# B&R Automation Studio project HealthCareDemo
Automation Studio 4.11.1.147; technology packages: mapp6D 1.1.10000, mappFramework 1.0.0, mappMotion 5.18.0, mappView 5.18.0

## Configuration 4PPC70

CPU 4PPC70.0573-20B, AutomationRuntime B4.91, Build 6.3.0, Safety 0.0, Vc V4.72.2

### Task classes (Cpu.sw)
```
Cyclic#1 (cycle 2000 us, tolerance 0 us):
  ConvSyncDe <- (binary)
  WaveDemo <- (binary)
  ConvUnload <- (binary)
  KalmanTes1 <- (binary)
  VariedMovD <- (binary)
  MacroDemo <- (binary)
  KalmanTest <- (binary)
  RoutingDem <- (binary)
  ProcSt2 <- (binary)
  ProcSt1 <- (binary)
  CycChlCfg <- (binary)
  InspectSt <- (binary)
  DofDemo <- (binary)
  ProcessDem <- (binary)
  DanceDemoC <- (binary)
Cyclic#8 (cycle 2000 us):
  RDICore <- Source.Core.RDICore.prg
DataObjects: McAcpSys
NcDataObjects: McDriveLog, AcpParTab
Binaries: udbdef, FWRules, mvLoader, mCoWebSc, TCData, arsvcreg, arflatprv, arcoal, TCLang, iomap, asfw, Role, ashwd, sysconf, arconfig, ashwac, User, TC, AssemConf, LayoutConf, CockpitSet, mcacpdrv, McAcpSim, McProfGen, McMechSys, MotConf, Hierarchy, VaxisConf, GroupConf, MechConf, FeatConf, AxisConf, FileConf, RecConf, Config_1, Config_2, OpcUaSrv, Config, Settings, CfgRecipe, CITT_FileU, CITT_Alarm, CITT_Recip, Config_4, Config_5, Config_3, Config_6, Config_8, Config_9, Config_7, Config_10, TraceConfi
Libraries: operator, runtime, astime, AsIecCon, McAcp6D, McBase, CoTrace, AsZip, FileIO, standard, AsBrStr, MpBase, MpRecipe, sys_lib, MpFile, brsystem, rdiAcp6D, arssl, asusb, dataobj, asmem, asio, asarprof, powerlnk, asepl, asarlog, aruser, McAcpTrak, MpAxis
```

### Hardware
```
4PPC70_0573_20B : 4PPC70.0573-20B v1.5.4.0
  Connector IF2:
    ActivateDevice = 1
    Mode = Manual
    InternetAddress = 192.168.10.10
    SubnetMask = 255.255.255.0
    ActivateSnmp = 2
    DeviceParam = /EDDN=gei
  ConfigurationID = OnsiteDemo_C80
  Simulation = 1
  UserRamSize = 15000
  RemMemSize = 15000
  RemanentGlobalPvSize = 1000
  TimerDeviceType = EPLX2X
  TimerDevice = 1685_CPU.IF1
  TaskClassIdleTime = 2000
  Cyclic1Duration = 2000
  Cyclic1Tolerance = 0
  Cyclic2Duration = 4000
  Cyclic2Tolerance = 4000
  Cyclic3Duration = 8000
  Cyclic3Tolerance = 8000
  Cyclic4Duration = 16000
  Cyclic4Tolerance = 16000
  Cyclic5Duration = 32000
  Cyclic5Tolerance = 32000
  Cyclic6Duration = 64000
  Cyclic6Tolerance = 64000
  Cyclic7Duration = 128000
  Cyclic7Tolerance = 128000
  Cyclic8Duration = 2000
  FileDevice1
  FileDeviceName1 = 6DMacro
  FileDevicePath1 = F:\Macros
  FileDevice2
  FileDeviceName2 = CNC_PrgDir
  FileDevicePath2 = F:/Programs/
  FileDevice3
  FileDeviceName3 = Recipe
  FileDevicePath3 = F:/Recipes/
  FileDevice4
  FileDeviceName4 = TeachFileDev
  FileDevicePath4 = F:/Teach/
  FileDevice5
  FileDeviceName5 = SvMovies
  FileDevicePath5 = F:/SvMovie
  FileDevice6
  FileDeviceName6 = User
  FileDevicePath6 = F:\
  FileDevice7
  FileDeviceName7 = 6DData
  FileDevicePath7 = C:\
  FtpUser1
  FtpUsername1 = bur  // user
  FtpUserPassword1 = kzPdX7T05qFX/2O0oq22KZRISpE2rDw4PeEeBt2Wff8=  // user
  FtpUserSalt1 = NaiTqhR1
  FTPAccessRight1 = 0
  FTPdevice1 = ALL
  ActivateOpcUa = 1
  OpcUaInformationModels_PV_Version = 1
  KeyMappingFile = VC\4PPC70_0573_20B.dis
8YFLM01.0000.00I-1 : 8YFLM01.0000.00I-1 v0.0.0.1
  Supervision = off
```

### IoMap.iom - 4PPC70_0573_20B/IoMap.iom
```iecst
VAR_CONFIG
	Cyclic#1.::gFB.In.Array[0] AT %IW."8YFLM01.0000.00I-1".EPL_FB_IN_0_I2007_S01;
	Cyclic#1.::gFB.In.Array[1] AT %IW."8YFLM01.0000.00I-1".EPL_FB_IN_1_I2007_S02;
	Cyclic#1.::gFB.In.Array[10] AT %IW."8YFLM01.0000.00I-1".EPL_FB_IN_10_I2007_S0B;
	Cyclic#1.::gFB.In.Array[100] AT %IW."8YFLM01.0000.00I-1".EPL_FB_IN_100_I2007_S65;
	Cyclic#1.::gFB.In.Array[101] AT %IW."8YFLM01.0000.00I-1".EPL_FB_IN_101_I2007_S66;
	Cyclic#1.::gFB.In.Array[102] AT %IW."8YFLM01.0000.00I-1".EPL_FB_IN_102_I2007_S67;
	Cyclic#1.::gFB.In.Array[103] AT %IW."8YFLM01.0000.00I-1".EPL_FB_IN_103_I2007_S68;
	Cyclic#1.::gFB.In.Array[104] AT %IW."8YFLM01.0000.00I-1".EPL_FB_IN_104_I2007_S69;
	Cyclic#1.::gFB.In.Array[105] AT %IW."8YFLM01.0000.00I-1".EPL_FB_IN_105_I2007_S6A;
	Cyclic#1.::gFB.In.Array[106] AT %IW."8YFLM01.0000.00I-1".EPL_FB_IN_106_I2007_S6B;
	Cyclic#1.::gFB.In.Array[107] AT %IW."8YFLM01.0000.00I-1".EPL_FB_IN_107_I2007_S6C;
	Cyclic#1.::gFB.In.Array[108] AT %IW."8YFLM01.0000.00I-1".EPL_FB_IN_108_I2007_S6D;
	Cyclic#1.::gFB.In.Array[109] AT %IW."8YFLM01.0000.00I-1".EPL_FB_IN_109_I2007_S6E;
	Cyclic#1.::gFB.In.Array[11] AT %IW."8YFLM01.0000.00I-1".EPL_FB_IN_11_I2007_S0C;
	Cyclic#1.::gFB.In.Array[110] AT %IW."8YFLM01.0000.00I-1".EPL_FB_IN_110_I2007_S6F;
	Cyclic#1.::gFB.In.Array[111] AT %IW."8YFLM01.0000.00I-1".EPL_FB_IN_111_I2007_S70;
	Cyclic#1.::gFB.In.Array[112] AT %IW."8YFLM01.0000.00I-1".EPL_FB_IN_112_I2007_S71;
	Cyclic#1.::gFB.In.Array[113] AT %IW."8YFLM01.0000.00I-1".EPL_FB_IN_113_I2007_S72;
	Cyclic#1.::gFB.In.Array[114] AT %IW."8YFLM01.0000.00I-1".EPL_FB_IN_114_I2007_S73;
	Cyclic#1.::gFB.In.Array[115] AT %IW."8YFLM01.0000.00I-1".EPL_FB_IN_115_I2007_S74;
	Cyclic#1.::gFB.In.Array[116] AT %IW."8YFLM01.0000.00I-1".EPL_FB_IN_116_I2007_S75;
	Cyclic#1.::gFB.In.Array[117] AT %IW."8YFLM01.0000.00I-1".EPL_FB_IN_117_I2007_S76;
	Cyclic#1.::gFB.In.Array[118] AT %IW."8YFLM01.0000.00I-1".EPL_FB_IN_118_I2007_S77;
	Cyclic#1.::gFB.In.Array[119] AT %IW."8YFLM01.0000.00I-1".EPL_FB_IN_119_I2007_S78;
	Cyclic#1.::gFB.In.Array[12] AT %IW."8YFLM01.0000.00I-1".EPL_FB_IN_12_I2007_S0D;
	Cyclic#1.::gFB.In.Array[120] AT %IW."8YFLM01.0000.00I-1".EPL_FB_IN_120_I2007_S79;
	Cyclic#1.::gFB.In.Array[121] AT %IW."8YFLM01.0000.00I-1".EPL_FB_IN_121_I2007_S7A;
	Cyclic#1.::gFB.In.Array[122] AT %IW."8YFLM01.0000.00I-1".EPL_FB_IN_122_I2007_S7B;
	Cyclic#1.::gFB.In.Array[123] AT %IW."8YFLM01.0000.00I-1".EPL_FB_IN_123_I2007_S7C;
	Cyclic#1.::gFB.In.Array[124] AT %IW."8YFLM01.0000.00I-1".EPL_FB_IN_124_I2007_S7D;
	Cyclic#1.::gFB.In.Array[125] AT %IW."8YFLM01.0000.00I-1".EPL_FB_IN_125_I2007_S7E;
	Cyclic#1.::gFB.In.Array[126] AT %IW."8YFLM01.0000.00I-1".EPL_FB_IN_126_I2007_S7F;
	Cyclic#1.::gFB.In.Array[127] AT %IW."8YFLM01.0000.00I-1".EPL_FB_IN_127_I2007_S80;
	Cyclic#1.::gFB.In.Array[128] AT %IW."8YFLM01.0000.00I-1".EPL_FB_IN_128_I2007_S81;
	Cyclic#1.::gFB.In.Array[129] AT %IW."8YFLM01.0000.00I-1".EPL_FB_IN_129_I2007_S82;
	Cyclic#1.::gFB.In.Array[13] AT %IW."8YFLM01.0000.00I-1".EPL_FB_IN_13_I2007_S0E;
	Cyclic#1.::gFB.In.Array[130] AT %IW."8YFLM01.0000.00I-1".EPL_FB_IN_130_I2007_S83;
	Cyclic#1.::gFB.In.Array[131] AT %IW."8YFLM01.0000.00I-1".EPL_FB_IN_131_I2007_S84;
	Cyclic#1.::gFB.In.Array[132] AT %IW."8YFLM01.0000.00I-1".EPL_FB_IN_132_I2007_S85;
	Cyclic#1.::gFB.In.Array[133] AT %IW."8YFLM01.0000.00I-1".EPL_FB_IN_133_I2007_S86;
	Cyclic#1.::gFB.In.Array[134] AT %IW."8YFLM01.0000.00I-1".EPL_FB_IN_134_I2007_S87;
	Cyclic#1.::gFB.In.Array[135] AT %IW."8YFLM01.0000.00I-1".EPL_FB_IN_135_I2007_S88;
	Cyclic#1.::gFB.In.Array[136] AT %IW."8YFLM01.0000.00I-1".EPL_FB_IN_136_I2007_S89;
	Cyclic#1.::gFB.In.Array[137] AT %IW."8YFLM01.0000.00I-1".EPL_FB_IN_137_I2007_S8A;
	Cyclic#1.::gFB.In.Array[138] AT %IW."8YFLM01.0000.00I-1".EPL_FB_IN_138_I2007_S8B;
	Cyclic#1.::gFB.In.Array[139] AT %IW."8YFLM01.0000.00I-1".EPL_FB_IN_139_I2007_S8C;
	Cyclic#1.::gFB.In.Array[14] AT %IW."8YFLM01.0000.00I-1".EPL_FB_IN_14_I2007_S0F;
	Cyclic#1.::gFB.In.Array[140] AT %IW."8YFLM01.0000.00I-1".EPL_FB_IN_140_I2007_S8D;
	Cyclic#1.::gFB.In.Array[141] AT %IW."8YFLM01.0000.00I-1".EPL_FB_IN_141_I2007_S8E;
	Cyclic#1.::gFB.In.Array[142] AT %IW."8YFLM01.0000.00I-1".EPL_FB_IN_142_I2007_S8F;
	Cyclic#1.::gFB.In.Array[143] AT %IW."8YFLM01.0000.00I-1".EPL_FB_IN_143_I2007_S90;
	Cyclic#1.::gFB.In.Array[144] AT %IW."8YFLM01.0000.00I-1".EPL_FB_IN_144_I2007_S91;
	Cyclic#1.::gFB.In.Array[145] AT %IW."8YFLM01.0000.00I-1".EPL_FB_IN_145_I2007_S92;
	Cyclic#1.::gFB.In.Array[146] AT %IW."8YFLM01.0000.00I-1".EPL_FB_IN_146_I2007_S93;
	Cyclic#1.::gFB.In.Array[147] AT %IW."8YFLM01.0000.00I-1".EPL_FB_IN_147_I2007_S94;
	Cyclic#1.::gFB.In.Array[148] AT %IW."8YFLM01.0000.00I-1".EPL_FB_IN_148_I2007_S95;
	Cyclic#1.::gFB.In.Array[149] AT %IW."8YFLM01.0000.00I-1".EPL_FB_IN_149_I2007_S96;
	Cyclic#1.::gFB.In.Array[15] AT %IW."8YFLM01.0000.00I-1".EPL_FB_IN_15_I2007_S10;
	Cyclic#1.::gFB.In.Array[150] AT %IW."8YFLM01.0000.00I-1".EPL_FB_IN_150_I2007_S97;
	Cyclic#1.::gFB.In.Array[151] AT %IW."8YFLM01.0000.00I-1".EPL_FB_IN_151_I2007_S98;
	Cyclic#1.::gFB.In.Array[152] AT %IW."8YFLM01.0000.00I-1".EPL_FB_IN_152_I2007_S99;
	Cyclic#1.::gFB.In.Array[153] AT %IW."8YFLM01.0000.00I-1".EPL_FB_IN_153_I2007_S9A;
	Cyclic#1.::gFB.In.Array[154] AT %IW."8YFLM01.0000.00I-1".EPL_FB_IN_154_I2007_S9B;
	Cyclic#1.::gFB.In.Array[155] AT %IW."8YFLM01.0000.00I-1".EPL_FB_IN_155_I2007_S9C;
	Cyclic#1.::gFB.In.Array[156] AT %IW."8YFLM01.0000.00I-1".EPL_FB_IN_156_I2007_S9D;
	Cyclic#1.::gFB.In.Array[157] AT %IW."8YFLM01.0000.00I-1".EPL_FB_IN_157_I2007_S9E;
	Cyclic#1.::gFB.In.Array[158] AT %IW."8YFLM01.0000.00I-1".EPL_FB_IN_158_I2007_S9F;
	Cyclic#1.::gFB.In.Array[159] AT %IW."8YFLM01.0000.00I-1".EPL_FB_IN_159_I2007_SA0;
	Cyclic#1.::gFB.In.Array[16] AT %IW."8YFLM01.0000.00I-1".EPL_FB_IN_16_I2007_S11;
	Cyclic#1.::gFB.In.Array[160] AT %IW."8YFLM01.0000.00I-1".EPL_FB_IN_160_I2007_SA1;
	Cyclic#1.::gFB.In.Array[161] AT %IW."8YFLM01.0000.00I-1".EPL_FB_IN_161_I2007_SA2;
	Cyclic#1.::gFB.In.Array[162] AT %IW."8YFLM01.0000.00I-1".EPL_FB_IN_162_I2007_SA3;
	Cyclic#1.::gFB.In.Array[163] AT %IW."8YFLM01.0000.00I-1".EPL_FB_IN_163_I2007_SA4;
	Cyclic#1.::gFB.In.Array[164] AT %IW."8YFLM01.0000.00I-1".EPL_FB_IN_164_I2007_SA5;
	Cyclic#1.::gFB.In.Array[165] AT %IW."8YFLM01.0000.00I-1".EPL_FB_IN_165_I2007_SA6;
	Cyclic#1.::gFB.In.Array[166] AT %IW."8YFLM01.0000.00I-1".EPL_FB_IN_166_I2007_SA7;
	Cyclic#1.::gFB.In.Array[167] AT %IW."8YFLM01.0000.00I-1".EPL_FB_IN_167_I2007_SA8;
	Cyclic#1.::gFB.In.Array[168] AT %IW."8YFLM01.0000.00I-1".EPL_FB_IN_168_I2007_SA9;
	Cyclic#1.::gFB.In.Array[169] AT %IW."8YFLM01.0000.00I-1".EPL_FB_IN_169_I2007_SAA;
	Cyclic#1.::gFB.In.Array[17] AT %IW."8YFLM01.0000.00I-1".EPL_FB_IN_17_I2007_S12;
	Cyclic#1.::gFB.In.Array[170] AT %IW."8YFLM01.0000.00I-1".EPL_FB_IN_170_I2007_SAB;
	Cyclic#1.::gFB.In.Array[171] AT %IW."8YFLM01.0000.00I-1".EPL_FB_IN_171_I2007_SAC;
	Cyclic#1.::gFB.In.Array[172] AT %IW."8YFLM01.0000.00I-1".EPL_FB_IN_172_I2007_SAD;
	Cyclic#1.::gFB.In.Array[173] AT %IW."8YFLM01.0000.00I-1".EPL_FB_IN_173_I2007_SAE;
	Cyclic#1.::gFB.In.Array[174] AT %IW."8YFLM01.0000.00I-1".EPL_FB_IN_174_I2007_SAF;
	Cyclic#1.::gFB.In.Array[175] AT %IW."8YFLM01.0000.00I-1".EPL_FB_IN_175_I2007_SB0;
	Cyclic#1.::gFB.In.Array[176] AT %IW."8YFLM01.0000.00I-1".EPL_FB_IN_176_I2007_SB1;
	Cyclic#1.::gFB.In.Array[177] AT %IW."8YFLM01.0000.00I-1".EPL_FB_IN_177_I2007_SB2;
	Cyclic#1.::gFB.In.Array[178] AT %IW."8YFLM01.0000.00I-1".EPL_FB_IN_178_I2007_SB3;
	Cyclic#1.::gFB.In.Array[179] AT %IW."8YFLM01.0000.00I-1".EPL_FB_IN_179_I2007_SB4;
	Cyclic#1.::gFB.In.Array[18] AT %IW."8YFLM01.0000.00I-1".EPL_FB_IN_18_I2007_S13;
	Cyclic#1.::gFB.In.Array[180] AT %IW."8YFLM01.0000.00I-1".EPL_FB_IN_180_I2007_SB5;
	Cyclic#1.::gFB.In.Array[181] AT %IW."8YFLM01.0000.00I-1".EPL_FB_IN_181_I2007_SB6;
	Cyclic#1.::gFB.In.Array[182] AT %IW."8YFLM01.0000.00I-1".EPL_FB_IN_182_I2007_SB7;
	Cyclic#1.::gFB.In.Array[183] AT %IW."8YFLM01.0000.00I-1".EPL_FB_IN_183_I2007_SB8;
	Cyclic#1.::gFB.In.Array[184] AT %IW."8YFLM01.0000.00I-1".EPL_FB_IN_184_I2007_SB9;
	Cyclic#1.::gFB.In.Array[185] AT %IW."8YFLM01.0000.00I-1".EPL_FB_IN_185_I2007_SBA;
	Cyclic#1.::gFB.In.Array[186] AT %IW."8YFLM01.0000.00I-1".EPL_FB_IN_186_I2007_SBB;
	Cyclic#1.::gFB.In.Array[187] AT %IW."8YFLM01.0000.00I-1".EPL_FB_IN_187_I2007_SBC;
	Cyclic#1.::gFB.In.Array[188] AT %IW."8YFLM01.0000.00I-1".EPL_FB_IN_188_I2007_SBD;
	Cyclic#1.::gFB.In.Array[189] AT %IW."8YFLM01.0000.00I-1".EPL_FB_IN_189_I2007_SBE;
	Cyclic#1.::gFB.In.Array[19] AT %IW."8YFLM01.0000.00I-1".EPL_FB_IN_19_I2007_S14;
	Cyclic#1.::gFB.In.Array[190] AT %IW."8YFLM01.0000.00I-1".EPL_FB_IN_190_I2007_SBF;
	Cyclic#1.::gFB.In.Array[191] AT %IW."8YFLM01.0000.00I-1".EPL_FB_IN_191_I2007_SC0;
	Cyclic#1.::gFB.In.Array[192] AT %IW."8YFLM01.0000.00I-1".EPL_FB_IN_192_I2007_SC1;
	Cyclic#1.::gFB.In.Array[193] AT %IW."8YFLM01.0000.00I-1".EPL_FB_IN_193_I2007_SC2;
	Cyclic#1.::gFB.In.Array[194] AT %IW."8YFLM01.0000.00I-1".EPL_FB_IN_194_I2007_SC3;
	Cyclic#1.::gFB.In.Array[195] AT %IW."8YFLM01.0000.00I-1".EPL_FB_IN_195_I2007_SC4;
	Cyclic#1.::gFB.In.Array[196] AT %IW."8YFLM01.0000.00I-1".EPL_FB_IN_196_I2007_SC5;
	Cyclic#1.::gFB.In.Array[197] AT %IW."8YFLM01.0000.00I-1".EPL_FB_IN_197_I2007_SC6;
	Cyclic#1.::gFB.In.Array[198] AT %IW."8YFLM01.0000.00I-1".EPL_FB_IN_198_I2007_SC7;
	Cyclic#1.::gFB.In.Array[199] AT %IW."8YFLM01.0000.00I-1".EPL_FB_IN_199_I2007_SC8;
	Cyclic#1.::gFB.In.Array[2] AT %IW."8YFLM01.0000.00I-1".EPL_FB_IN_2_I2007_S03;
	Cyclic#1.::gFB.In.Array[20] AT %IW."8YFLM01.0000.00I-1".EPL_FB_IN_20_I2007_S15;
	Cyclic#1.::gFB.In.Array[21] AT %IW."8YFLM01.0000.00I-1".EPL_FB_IN_21_I2007_S16;
	Cyclic#1.::gFB.In.Array[22] AT %IW."8YFLM01.0000.00I-1".EPL_FB_IN_22_I2007_S17;
	Cyclic#1.::gFB.In.Array[23] AT %IW."8YFLM01.0000.00I-1".EPL_FB_IN_23_I2007_S18;
	Cyclic#1.::gFB.In.Array[24] AT %IW."8YFLM01.0000.00I-1".EPL_FB_IN_24_I2007_S19;
	Cyclic#1.::gFB.In.Array[25] AT %IW."8YFLM01.0000.00I-1".EPL_FB_IN_25_I2007_S1A;
	Cyclic#1.::gFB.In.Array[26] AT %IW."8YFLM01.0000.00I-1".EPL_FB_IN_26_I2007_S1B;
	Cyclic#1.::gFB.In.Array[27] AT %IW."8YFLM01.0000.00I-1".EPL_FB_IN_27_I2007_S1C;
	Cyclic#1.::gFB.In.Array[28] AT %IW."8YFLM01.0000.00I-1".EPL_FB_IN_28_I2007_S1D;
	Cyclic#1.::gFB.In.Array[29] AT %IW."8YFLM01.0000.00I-1".EPL_FB_IN_29_I2007_S1E;
	Cyclic#1.::gFB.In.Array[3] AT %IW."8YFLM01.0000.00I-1".EPL_FB_IN_3_I2007_S04;
	Cyclic#1.::gFB.In.Array[30] AT %IW."8YFLM01.0000.00I-1".EPL_FB_IN_30_I2007_S1F;
	Cyclic#1.::gFB.In.Array[31] AT %IW."8YFLM01.0000.00I-1".EPL_FB_IN_31_I2007_S20;
	Cyclic#1.::gFB.In.Array[32] AT %IW."8YFLM01.0000.00I-1".EPL_FB_IN_32_I2007_S21;
	Cyclic#1.::gFB.In.Array[33] AT %IW."8YFLM01.0000.00I-1".EPL_FB_IN_33_I2007_S22;
	Cyclic#1.::gFB.In.Array[34] AT %IW."8YFLM01.0000.00I-1".EPL_FB_IN_34_I2007_S23;
	Cyclic#1.::gFB.In.Array[35] AT %IW."8YFLM01.0000.00I-1".EPL_FB_IN_35_I2007_S24;
	Cyclic#1.::gFB.In.Array[36] AT %IW."8YFLM01.0000.00I-1".EPL_FB_IN_36_I2007_S25;
	Cyclic#1.::gFB.In.Array[37] AT %IW."8YFLM01.0000.00I-1".EPL_FB_IN_37_I2007_S26;
	Cyclic#1.::gFB.In.Array[38] AT %IW."8YFLM01.0000.00I-1".EPL_FB_IN_38_I2007_S27;
	Cyclic#1.::gFB.In.Array[39] AT %IW."8YFLM01.0000.00I-1".EPL_FB_IN_39_I2007_S28;
	Cyclic#1.::gFB.In.Array[4] AT %IW."8YFLM01.0000.00I-1".EPL_FB_IN_4_I2007_S05;
	Cyclic#1.::gFB.In.Array[40] AT %IW."8YFLM01.0000.00I-1".EPL_FB_IN_40_I2007_S29;
	Cyclic#1.::gFB.In.Array[41] AT %IW."8YFLM01.0000.00I-1".EPL_FB_IN_41_I2007_S2A;
	Cyclic#1.::gFB.In.Array[42] AT %IW."8YFLM01.0000.00I-1".EPL_FB_IN_42_I2007_S2B;
	Cyclic#1.::gFB.In.Array[43] AT %IW."8YFLM01.0000.00I-1".EPL_FB_IN_43_I2007_S2C;
	Cyclic#1.::gFB.In.Array[44] AT %IW."8YFLM01.0000.00I-1".EPL_FB_IN_44_I2007_S2D;
	Cyclic#1.::gFB.In.Array[45] AT %IW."8YFLM01.0000.00I-1".EPL_FB_IN_45_I2007_S2E;
	Cyclic#1.::gFB.In.Array[46] AT %IW."8YFLM01.0000.00I-1".EPL_FB_IN_46_I2007_S2F;
	Cyclic#1.::gFB.In.Array[47] AT %IW."8YFLM01.0000.00I-1".EPL_FB_IN_47_I2007_S30;
	Cyclic#1.::gFB.In.Array[48] AT %IW."8YFLM01.0000.00I-1".EPL_FB_IN_48_I2007_S31;
	Cyclic#1.::gFB.In.Array[49] AT %IW."8YFLM01.0000.00I-1".EPL_FB_IN_49_I2007_S32;
	Cyclic#1.::gFB.In.Array[5] AT %IW."8YFLM01.0000.00I-1".EPL_FB_IN_5_I2007_S06;
	Cyclic#1.::gFB.In.Array[50] AT %IW."8YFLM01.0000.00I-1".EPL_FB_IN_50_I2007_S33;
	Cyclic#1.::gFB.In.Array[51] AT %IW."8YFLM01.0000.00I-1".EPL_FB_IN_51_I2007_S34;
	Cyclic#1.::gFB.In.Array[52] AT %IW."8YFLM01.0000.00I-1".EPL_FB_IN_52_I2007_S35;
	Cyclic#1.::gFB.In.Array[53] AT %IW."8YFLM01.0000.00I-1".EPL_FB_IN_53_I2007_S36;
	Cyclic#1.::gFB.In.Array[54] AT %IW."8YFLM01.0000.00I-1".EPL_FB_IN_54_I2007_S37;
	Cyclic#1.::gFB.In.Array[55] AT %IW."8YFLM01.0000.00I-1".EPL_FB_IN_55_I2007_S38;
	Cyclic#1.::gFB.In.Array[56] AT %IW."8YFLM01.0000.00I-1".EPL_FB_IN_56_I2007_S39;
	Cyclic#1.::gFB.In.Array[57] AT %IW."8YFLM01.0000.00I-1".EPL_FB_IN_57_I2007_S3A;
	Cyclic#1.::gFB.In.Array[58] AT %IW."8YFLM01.0000.00I-1".EPL_FB_IN_58_I2007_S3B;
	Cyclic#1.::gFB.In.Array[59] AT %IW."8YFLM01.0000.00I-1".EPL_FB_IN_59_I2007_S3C;
	Cyclic#1.::gFB.In.Array[6] AT %IW."8YFLM01.0000.00I-1".EPL_FB_IN_6_I2007_S07;
	Cyclic#1.::gFB.In.Array[60] AT %IW."8YFLM01.0000.00I-1".EPL_FB_IN_60_I2007_S3D;
	Cyclic#1.::gFB.In.Array[61] AT %IW."8YFLM01.0000.00I-1".EPL_FB_IN_61_I2007_S3E;
	Cyclic#1.::gFB.In.Array[62] AT %IW."8YFLM01.0000.00I-1".EPL_FB_IN_62_I2007_S3F;
	Cyclic#1.::gFB.In.Array[63] AT %IW."8YFLM01.0000.00I-1".EPL_FB_IN_63_I2007_S40;
	Cyclic#1.::gFB.In.Array[64] AT %IW."8YFLM01.0000.00I-1".EPL_FB_IN_64_I2007_S41;
	Cyclic#1.::gFB.In.Array[65] AT %IW."8YFLM01.0000.00I-1".EPL_FB_IN_65_I2007_S42;
	Cyclic#1.::gFB.In.Array[66] AT %IW."8YFLM01.0000.00I-1".EPL_FB_IN_66_I2007_S43;
	Cyclic#1.::gFB.In.Array[67] AT %IW."8YFLM01.0000.00I-1".EPL_FB_IN_67_I2007_S44;
	Cyclic#1.::gFB.In.Array[68] AT %IW."8YFLM01.0000.00I-1".EPL_FB_IN_68_I2007_S45;
	Cyclic#1.::gFB.In.Array[69] AT %IW."8YFLM01.0000.00I-1".EPL_FB_IN_69_I2007_S46;
	Cyclic#1.::gFB.In.Array[7] AT %IW."8YFLM01.0000.00I-1".EPL_FB_IN_7_I2007_S08;
	Cyclic#1.::gFB.In.Array[70] AT %IW."8YFLM01.0000.00I-1".EPL_FB_IN_70_I2007_S47;
	Cyclic#1.::gFB.In.Array[71] AT %IW."8YFLM01.0000.00I-1".EPL_FB_IN_71_I2007_S48;
	Cyclic#1.::gFB.In.Array[72] AT %IW."8YFLM01.0000.00I-1".EPL_FB_IN_72_I2007_S49;
	Cyclic#1.::gFB.In.Array[73] AT %IW."8YFLM01.0000.00I-1".EPL_FB_IN_73_I2007_S4A;
	Cyclic#1.::gFB.In.Array[74] AT %IW."8YFLM01.0000.00I-1".EPL_FB_IN_74_I2007_S4B;
	Cyclic#1.::gFB.In.Array[75] AT %IW."8YFLM01.0000.00I-1".EPL_FB_IN_75_I2007_S4C;
	Cyclic#1.::gFB.In.Array[76] AT %IW."8YFLM01.0000.00I-1".EPL_FB_IN_76_I2007_S4D;
	Cyclic#1.::gFB.In.Array[77] AT %IW."8YFLM01.0000.00I-1".EPL_FB_IN_77_I2007_S4E;
	Cyclic#1.::gFB.In.Array[78] AT %IW."8YFLM01.0000.00I-1".EPL_FB_IN_78_I2007_S4F;
	Cyclic#1.::gFB.In.Array[79] AT %IW."8YFLM01.0000.00I-1".EPL_FB_IN_79_I2007_S50;
	Cyclic#1.::gFB.In.Array[8] AT %IW."8YFLM01.0000.00I-1".EPL_FB_IN_8_I2007_S09;
	Cyclic#1.::gFB.In.Array[80] AT %IW."8YFLM01.0000.00I-1".EPL_FB_IN_80_I2007_S51;
	Cyclic#1.::gFB.In.Array[81] AT %IW."8YFLM01.0000.00I-1".EPL_FB_IN_81_I2007_S52;
	Cyclic#1.::gFB.In.Array[82] AT %IW."8YFLM01.0000.00I-1".EPL_FB_IN_82_I2007_S53;
	Cyclic#1.::gFB.In.Array[83] AT %IW."8YFLM01.0000.00I-1".EPL_FB_IN_83_I2007_S54;
	Cyclic#1.::gFB.In.Array[84] AT %IW."8YFLM01.0000.00I-1".EPL_FB_IN_84_I2007_S55;
	Cyclic#1.::gFB.In.Array[85] AT %IW."8YFLM01.0000.00I-1".EPL_FB_IN_85_I2007_S56;
	Cyclic#1.::gFB.In.Array[86] AT %IW."8YFLM01.0000.00I-1".EPL_FB_IN_86_I2007_S57;
	Cyclic#1.::gFB.In.Array[87] AT %IW."8YFLM01.0000.00I-1".EPL_FB_IN_87_I2007_S58;
	Cyclic#1.::gFB.In.Array[88] AT %IW."8YFLM01.0000.00I-1".EPL_FB_IN_88_I2007_S59;
	Cyclic#1.::gFB.In.Array[89] AT %IW."8YFLM01.0000.00I-1".EPL_FB_IN_89_I2007_S5A;
	Cyclic#1.::gFB.In.Array[9] AT %IW."8YFLM01.0000.00I-1".EPL_FB_IN_9_I2007_S0A;
	Cyclic#1.::gFB.In.Array[90] AT %IW."8YFLM01.0000.00I-1".EPL_FB_IN_90_I2007_S5B;
	Cyclic#1.::gFB.In.Array[91] AT %IW."8YFLM01.0000.00I-1".EPL_FB_IN_91_I2007_S5C;
	Cyclic#1.::gFB.In.Array[92] AT %IW."8YFLM01.0000.00I-1".EPL_FB_IN_92_I2007_S5D;
	Cyclic#1.::gFB.In.Array[93] AT %IW."8YFLM01.0000.00I-1".EPL_FB_IN_93_I2007_S5E;
	Cyclic#1.::gFB.In.Array[94] AT %IW."8YFLM01.0000.00I-1".EPL_FB_IN_94_I2007_S5F;
	Cyclic#1.::gFB.In.Array[95] AT %IW."8YFLM01.0000.00I-1".EPL_FB_IN_95_I2007_S60;
	Cyclic#1.::gFB.In.Array[96] AT %IW."8YFLM01.0000.00I-1".EPL_FB_IN_96_I2007_S61;
	Cyclic#1.::gFB.In.Array[97] AT %IW."8YFLM01.0000.00I-1".EPL_FB_IN_97_I2007_S62;
	Cyclic#1.::gFB.In.Array[98] AT %IW."8YFLM01.0000.00I-1".EPL_FB_IN_98_I2007_S63;
	Cyclic#1.::gFB.In.Array[99] AT %IW."8YFLM01.0000.00I-1".EPL_FB_IN_99_I2007_S64;
	Cyclic#1.::gFB.Out.Array[0] AT %QW."8YFLM01.0000.00I-1".EPL_FB_OUT_0_I2008_S01Out;
	Cyclic#1.::gFB.Out.Array[1] AT %QW."8YFLM01.0000.00I-1".EPL_FB_OUT_1_I2008_S02Out;
	Cyclic#1.::gFB.Out.Array[10] AT %QW."8YFLM01.0000.00I-1".EPL_FB_OUT_10_I2008_S0BOut;
	Cyclic#1.::gFB.Out.Array[100] AT %QW."8YFLM01.0000.00I-1".EPL_FB_OUT_100_I2008_S65Out;
	Cyclic#1.::gFB.Out.Array[101] AT %QW."8YFLM01.0000.00I-1".EPL_FB_OUT_101_I2008_S66Out;
	Cyclic#1.::gFB.Out.Array[102] AT %QW."8YFLM01.0000.00I-1".EPL_FB_OUT_102_I2008_S67Out;
	Cyclic#1.::gFB.Out.Array[103] AT %QW."8YFLM01.0000.00I-1".EPL_FB_OUT_103_I2008_S68Out;
	Cyclic#1.::gFB.Out.Array[104] AT %QW."8YFLM01.0000.00I-1".EPL_FB_OUT_104_I2008_S69Out;
	Cyclic#1.::gFB.Out.Array[105] AT %QW."8YFLM01.0000.00I-1".EPL_FB_OUT_105_I2008_S6AOut;
	Cyclic#1.::gFB.Out.Array[106] AT %QW."8YFLM01.0000.00I-1".EPL_FB_OUT_106_I2008_S6BOut;
	Cyclic#1.::gFB.Out.Array[107] AT %QW."8YFLM01.0000.00I-1".EPL_FB_OUT_107_I2008_S6COut;
	Cyclic#1.::gFB.Out.Array[108] AT %QW."8YFLM01.0000.00I-1".EPL_FB_OUT_108_I2008_S6DOut;
	Cyclic#1.::gFB.Out.Array[109] AT %QW."8YFLM01.0000.00I-1".EPL_FB_OUT_109_I2008_S6EOut;
	Cyclic#1.::gFB.Out.Array[11] AT %QW."8YFLM01.0000.00I-1".EPL_FB_OUT_11_I2008_S0COut;
	Cyclic#1.::gFB.Out.Array[110] AT %QW."8YFLM01.0000.00I-1".EPL_FB_OUT_110_I2008_S6FOut;
	Cyclic#1.::gFB.Out.Array[111] AT %QW."8YFLM01.0000.00I-1".EPL_FB_OUT_111_I2008_S70Out;
	Cyclic#1.::gFB.Out.Array[112] AT %QW."8YFLM01.0000.00I-1".EPL_FB_OUT_112_I2008_S71Out;
	Cyclic#1.::gFB.Out.Array[113] AT %QW."8YFLM01.0000.00I-1".EPL_FB_OUT_113_I2008_S72Out;
	Cyclic#1.::gFB.Out.Array[114] AT %QW."8YFLM01.0000.00I-1".EPL_FB_OUT_114_I2008_S73Out;
	Cyclic#1.::gFB.Out.Array[115] AT %QW."8YFLM01.0000.00I-1".EPL_FB_OUT_115_I2008_S74Out;
	Cyclic#1.::gFB.Out.Array[116] AT %QW."8YFLM01.0000.00I-1".EPL_FB_OUT_116_I2008_S75Out;
	Cyclic#1.::gFB.Out.Array[117] AT %QW."8YFLM01.0000.00I-1".EPL_FB_OUT_117_I2008_S76Out;
	Cyclic#1.::gFB.Out.Array[118] AT %QW."8YFLM01.0000.00I-1".EPL_FB_OUT_118_I2008_S77Out;
	Cyclic#1.::gFB.Out.Array[119] AT %QW."8YFLM01.0000.00I-1".EPL_FB_OUT_119_I2008_S78Out;
	Cyclic#1.::gFB.Out.Array[12] AT %QW."8YFLM01.0000.00I-1".EPL_FB_OUT_12_I2008_S0DOut;
	Cyclic#1.::gFB.Out.Array[120] AT %QW."8YFLM01.0000.00I-1".EPL_FB_OUT_120_I2008_S79Out;
	Cyclic#1.::gFB.Out.Array[121] AT %QW."8YFLM01.0000.00I-1".EPL_FB_OUT_121_I2008_S7AOut;
	Cyclic#1.::gFB.Out.Array[122] AT %QW."8YFLM01.0000.00I-1".EPL_FB_OUT_122_I2008_S7BOut;
	Cyclic#1.::gFB.Out.Array[123] AT %QW."8YFLM01.0000.00I-1".EPL_FB_OUT_123_I2008_S7COut;
	Cyclic#1.::gFB.Out.Array[124] AT %QW."8YFLM01.0000.00I-1".EPL_FB_OUT_124_I2008_S7DOut;
	Cyclic#1.::gFB.Out.Array[125] AT %QW."8YFLM01.0000.00I-1".EPL_FB_OUT_125_I2008_S7EOut;
	Cyclic#1.::gFB.Out.Array[126] AT %QW."8YFLM01.0000.00I-1".EPL_FB_OUT_126_I2008_S7FOut;
	Cyclic#1.::gFB.Out.Array[127] AT %QW."8YFLM01.0000.00I-1".EPL_FB_OUT_127_I2008_S80Out;
	Cyclic#1.::gFB.Out.Array[128] AT %QW."8YFLM01.0000.00I-1".EPL_FB_OUT_128_I2008_S81Out;
	Cyclic#1.::gFB.Out.Array[129] AT %QW."8YFLM01.0000.00I-1".EPL_FB_OUT_129_I2008_S82Out;
	Cyclic#1.::gFB.Out.Array[13] AT %QW."8YFLM01.0000.00I-1".EPL_FB_OUT_13_I2008_S0EOut;
	Cyclic#1.::gFB.Out.Array[130] AT %QW."8YFLM01.0000.00I-1".EPL_FB_OUT_130_I2008_S83Out;
	Cyclic#1.::gFB.Out.Array[131] AT %QW."8YFLM01.0000.00I-1".EPL_FB_OUT_131_I2008_S84Out;
	Cyclic#1.::gFB.Out.Array[132] AT %QW."8YFLM01.0000.00I-1".EPL_FB_OUT_132_I2008_S85Out;
	Cyclic#1.::gFB.Out.Array[133] AT %QW."8YFLM01.0000.00I-1".EPL_FB_OUT_133_I2008_S86Out;
	Cyclic#1.::gFB.Out.Array[134] AT %QW."8YFLM01.0000.00I-1".EPL_FB_OUT_134_I2008_S87Out;
	Cyclic#1.::gFB.Out.Array[135] AT %QW."8YFLM01.0000.00I-1".EPL_FB_OUT_135_I2008_S88Out;
	Cyclic#1.::gFB.Out.Array[136] AT %QW."8YFLM01.0000.00I-1".EPL_FB_OUT_136_I2008_S89Out;
	Cyclic#1.::gFB.Out.Array[137] AT %QW."8YFLM01.0000.00I-1".EPL_FB_OUT_137_I2008_S8AOut;
	Cyclic#1.::gFB.Out.Array[138] AT %QW."8YFLM01.0000.00I-1".EPL_FB_OUT_138_I2008_S8BOut;
	Cyclic#1.::gFB.Out.Array[139] AT %QW."8YFLM01.0000.00I-1".EPL_FB_OUT_139_I2008_S8COut;
	Cyclic#1.::gFB.Out.Array[14] AT %QW."8YFLM01.0000.00I-1".EPL_FB_OUT_14_I2008_S0FOut;
	Cyclic#1.::gFB.Out.Array[140] AT %QW."8YFLM01.0000.00I-1".EPL_FB_OUT_140_I2008_S8DOut;
	Cyclic#1.::gFB.Out.Array[141] AT %QW."8YFLM01.0000.00I-1".EPL_FB_OUT_141_I2008_S8EOut;
	Cyclic#1.::gFB.Out.Array[142] AT %QW."8YFLM01.0000.00I-1".EPL_FB_OUT_142_I2008_S8FOut;
	Cyclic#1.::gFB.Out.Array[143] AT %QW."8YFLM01.0000.00I-1".EPL_FB_OUT_143_I2008_S90Out;
	Cyclic#1.::gFB.Out.Array[144] AT %QW."8YFLM01.0000.00I-1".EPL_FB_OUT_144_I2008_S91Out;
	Cyclic#1.::gFB.Out.Array[145] AT %QW."8YFLM01.0000.00I-1".EPL_FB_OUT_145_I2008_S92Out;
	Cyclic#1.::gFB.Out.Array[146] AT %QW."8YFLM01.0000.00I-1".EPL_FB_OUT_146_I2008_S93Out;
	Cyclic#1.::gFB.Out.Array[147] AT %QW."8YFLM01.0000.00I-1".EPL_FB_OUT_147_I2008_S94Out;
	Cyclic#1.::gFB.Out.Array[148] AT %QW."8YFLM01.0000.00I-1".EPL_FB_OUT_148_I2008_S95Out;
	Cyclic#1.::gFB.Out.Array[149] AT %QW."8YFLM01.0000.00I-1".EPL_FB_OUT_149_I2008_S96Out;
	Cyclic#1.::gFB.Out.Array[15] AT %QW."8YFLM01.0000.00I-1".EPL_FB_OUT_15_I2008_S10Out;
	Cyclic#1.::gFB.Out.Array[150] AT %QW."8YFLM01.0000.00I-1".EPL_FB_OUT_150_I2008_S97Out;
	Cyclic#1.::gFB.Out.Array[151] AT %QW."8YFLM01.0000.00I-1".EPL_FB_OUT_151_I2008_S98Out;
	Cyclic#1.::gFB.Out.Array[152] AT %QW."8YFLM01.0000.00I-1".EPL_FB_OUT_152_I2008_S99Out;
	Cyclic#1.::gFB.Out.Array[153] AT %QW."8YFLM01.0000.00I-1".EPL_FB_OUT_153_I2008_S9AOut;
	Cyclic#1.::gFB.Out.Array[154] AT %QW."8YFLM01.0000.00I-1".EPL_FB_OUT_154_I2008_S9BOut;
	Cyclic#1.::gFB.Out.Array[155] AT %QW."8YFLM01.0000.00I-1".EPL_FB_OUT_155_I2008_S9COut;
	Cyclic#1.::gFB.Out.Array[156] AT %QW."8YFLM01.0000.00I-1".EPL_FB_OUT_156_I2008_S9DOut;
	Cyclic#1.::gFB.Out.Array[157] AT %QW."8YFLM01.0000.00I-1".EPL_FB_OUT_157_I2008_S9EOut;
	Cyclic#1.::gFB.Out.Array[158] AT %QW."8YFLM01.0000.00I-1".EPL_FB_OUT_158_I2008_S9FOut;
	Cyclic#1.::gFB.Out.Array[159] AT %QW."8YFLM01.0000.00I-1".EPL_FB_OUT_159_I2008_SA0Out;
	Cyclic#1.::gFB.Out.Array[16] AT %QW."8YFLM01.0000.00I-1".EPL_FB_OUT_16_I2008_S11Out;
	Cyclic#1.::gFB.Out.Array[160] AT %QW."8YFLM01.0000.00I-1".EPL_FB_OUT_160_I2008_SA1Out;
	Cyclic#1.::gFB.Out.Array[161] AT %QW."8YFLM01.0000.00I-1".EPL_FB_OUT_161_I2008_SA2Out;
	Cyclic#1.::gFB.Out.Array[162] AT %QW."8YFLM01.0000.00I-1".EPL_FB_OUT_162_I2008_SA3Out;
	Cyclic#1.::gFB.Out.Array[163] AT %QW."8YFLM01.0000.00I-1".EPL_FB_OUT_163_I2008_SA4Out;
	Cyclic#1.::gFB.Out.Array[164] AT %QW."8YFLM01.0000.00I-1".EPL_FB_OUT_164_I2008_SA5Out;
	Cyclic#1.::gFB.Out.Array[165] AT %QW."8YFLM01.0000.00I-1".EPL_FB_OUT_165_I2008_SA6Out;
	Cyclic#1.::gFB.Out.Array[166] AT %QW."8YFLM01.0000.00I-1".EPL_FB_OUT_166_I2008_SA7Out;
	Cyclic#1.::gFB.Out.Array[167] AT %QW."8YFLM01.0000.00I-1".EPL_FB_OUT_167_I2008_SA8Out;
	Cyclic#1.::gFB.Out.Array[168] AT %QW."8YFLM01.0000.00I-1".EPL_FB_OUT_168_I2008_SA9Out;
	Cyclic#1.::gFB.Out.Array[169] AT %QW."8YFLM01.0000.00I-1".EPL_FB_OUT_169_I2008_SAAOut;
	Cyclic#1.::gFB.Out.Array[17] AT %QW."8YFLM01.0000.00I-1".EPL_FB_OUT_17_I2008_S12Out;
	Cyclic#1.::gFB.Out.Array[170] AT %QW."8YFLM01.0000.00I-1".EPL_FB_OUT_170_I2008_SABOut;
	Cyclic#1.::gFB.Out.Array[171] AT %QW."8YFLM01.0000.00I-1".EPL_FB_OUT_171_I2008_SACOut;
	Cyclic#1.::gFB.Out.Array[172] AT %QW."8YFLM01.0000.00I-1".EPL_FB_OUT_172_I2008_SADOut;
	Cyclic#1.::gFB.Out.Array[173] AT %QW."8YFLM01.0000.00I-1".EPL_FB_OUT_173_I2008_SAEOut;
	Cyclic#1.::gFB.Out.Array[174] AT %QW."8YFLM01.0000.00I-1".EPL_FB_OUT_174_I2008_SAFOut;
	Cyclic#1.::gFB.Out.Array[175] AT %QW."8YFLM01.0000.00I-1".EPL_FB_OUT_175_I2008_SB0Out;
	Cyclic#1.::gFB.Out.Array[176] AT %QW."8YFLM01.0000.00I-1".EPL_FB_OUT_176_I2008_SB1Out;
	Cyclic#1.::gFB.Out.Array[177] AT %QW."8YFLM01.0000.00I-1".EPL_FB_OUT_177_I2008_SB2Out;
	Cyclic#1.::gFB.Out.Array[178] AT %QW."8YFLM01.0000.00I-1".EPL_FB_OUT_178_I2008_SB3Out;
	Cyclic#1.::gFB.Out.Array[179] AT %QW."8YFLM01.0000.00I-1".EPL_FB_OUT_179_I2008_SB4Out;
	Cyclic#1.::gFB.Out.Array[18] AT %QW."8YFLM01.0000.00I-1".EPL_FB_OUT_18_I2008_S13Out;
	Cyclic#1.::gFB.Out.Array[180] AT %QW."8YFLM01.0000.00I-1".EPL_FB_OUT_180_I2008_SB5Out;
	Cyclic#1.::gFB.Out.Array[181] AT %QW."8YFLM01.0000.00I-1".EPL_FB_OUT_181_I2008_SB6Out;
	Cyclic#1.::gFB.Out.Array[182] AT %QW."8YFLM01.0000.00I-1".EPL_FB_OUT_182_I2008_SB7Out;
	Cyclic#1.::gFB.Out.Array[183] AT %QW."8YFLM01.0000.00I-1".EPL_FB_OUT_183_I2008_SB8Out;
	Cyclic#1.::gFB.Out.Array[184] AT %QW."8YFLM01.0000.00I-1".EPL_FB_OUT_184_I2008_SB9Out;
	Cyclic#1.::gFB.Out.Array[185] AT %QW."8YFLM01.0000.00I-1".EPL_FB_OUT_185_I2008_SBAOut;
	Cyclic#1.::gFB.Out.Array[186] AT %QW."8YFLM01.0000.00I-1".EPL_FB_OUT_186_I2008_SBBOut;
	Cyclic#1.::gFB.Out.Array[187] AT %QW."8YFLM01.0000.00I-1".EPL_FB_OUT_187_I2008_SBCOut;
	Cyclic#1.::gFB.Out.Array[188] AT %QW."8YFLM01.0000.00I-1".EPL_FB_OUT_188_I2008_SBDOut;
	Cyclic#1.::gFB.Out.Array[189] AT %QW."8YFLM01.0000.00I-1".EPL_FB_OUT_189_I2008_SBEOut;
	Cyclic#1.::gFB.Out.Array[19] AT %QW."8YFLM01.0000.00I-1".EPL_FB_OUT_19_I2008_S14Out;
	Cyclic#1.::gFB.Out.Array[190] AT %QW."8YFLM01.0000.00I-1".EPL_FB_OUT_190_I2008_SBFOut;
	Cyclic#1.::gFB.Out.Array[191] AT %QW."8YFLM01.0000.00I-1".EPL_FB_OUT_191_I2008_SC0Out;
	Cyclic#1.::gFB.Out.Array[192] AT %QW."8YFLM01.0000.00I-1".EPL_FB_OUT_192_I2008_SC1Out;
	Cyclic#1.::gFB.Out.Array[193] AT %QW."8YFLM01.0000.00I-1".EPL_FB_OUT_193_I2008_SC2Out;
	Cyclic#1.::gFB.Out.Array[194] AT %QW."8YFLM01.0000.00I-1".EPL_FB_OUT_194_I2008_SC3Out;
	Cyclic#1.::gFB.Out.Array[195] AT %QW."8YFLM01.0000.00I-1".EPL_FB_OUT_195_I2008_SC4Out;
	Cyclic#1.::gFB.Out.Array[196] AT %QW."8YFLM01.0000.00I-1".EPL_FB_OUT_196_I2008_SC5Out;
	Cyclic#1.::gFB.Out.Array[197] AT %QW."8YFLM01.0000.00I-1".EPL_FB_OUT_197_I2008_SC6Out;
	Cyclic#1.::gFB.Out.Array[198] AT %QW."8YFLM01.0000.00I-1".EPL_FB_OUT_198_I2008_SC7Out;
	Cyclic#1.::gFB.Out.Array[199] AT %QW."8YFLM01.0000.00I-1".EPL_FB_OUT_199_I2008_SC8Out;
	Cyclic#1.::gFB.Out.Array[2] AT %QW."8YFLM01.0000.00I-1".EPL_FB_OUT_2_I2008_S03Out;
	Cyclic#1.::gFB.Out.Array[20] AT %QW."8YFLM01.0000.00I-1".EPL_FB_OUT_20_I2008_S15Out;
	Cyclic#1.::gFB.Out.Array[21] AT %QW."8YFLM01.0000.00I-1".EPL_FB_OUT_21_I2008_S16Out;
	Cyclic#1.::gFB.Out.Array[22] AT %QW."8YFLM01.0000.00I-1".EPL_FB_OUT_22_I2008_S17Out;
	Cyclic#1.::gFB.Out.Array[23] AT %QW."8YFLM01.0000.00I-1".EPL_FB_OUT_23_I2008_S18Out;
	Cyclic#1.::gFB.Out.Array[24] AT %QW."8YFLM01.0000.00I-1".EPL_FB_OUT_24_I2008_S19Out;
	Cyclic#1.::gFB.Out.Array[25] AT %QW."8YFLM01.0000.00I-1".EPL_FB_OUT_25_I2008_S1AOut;
	Cyclic#1.::gFB.Out.Array[26] AT %QW."8YFLM01.0000.00I-1".EPL_FB_OUT_26_I2008_S1BOut;
	Cyclic#1.::gFB.Out.Array[27] AT %QW."8YFLM01.0000.00I-1".EPL_FB_OUT_27_I2008_S1COut;
	Cyclic#1.::gFB.Out.Array[28] AT %QW."8YFLM01.0000.00I-1".EPL_FB_OUT_28_I2008_S1DOut;
	Cyclic#1.::gFB.Out.Array[29] AT %QW."8YFLM01.0000.00I-1".EPL_FB_OUT_29_I2008_S1EOut;
	Cyclic#1.::gFB.Out.Array[3] AT %QW."8YFLM01.0000.00I-1".EPL_FB_OUT_3_I2008_S04Out;
	Cyclic#1.::gFB.Out.Array[30] AT %QW."8YFLM01.0000.00I-1".EPL_FB_OUT_30_I2008_S1FOut;
	Cyclic#1.::gFB.Out.Array[31] AT %QW."8YFLM01.0000.00I-1".EPL_FB_OUT_31_I2008_S20Out;
	Cyclic#1.::gFB.Out.Array[32] AT %QW."8YFLM01.0000.00I-1".EPL_FB_OUT_32_I2008_S21Out;
	Cyclic#1.::gFB.Out.Array[33] AT %QW."8YFLM01.0000.00I-1".EPL_FB_OUT_33_I2008_S22Out;
	Cyclic#1.::gFB.Out.Array[34] AT %QW."8YFLM01.0000.00I-1".EPL_FB_OUT_34_I2008_S23Out;
	Cyclic#1.::gFB.Out.Array[35] AT %QW."8YFLM01.0000.00I-1".EPL_FB_OUT_35_I2008_S24Out;
	Cyclic#1.::gFB.Out.Array[36] AT %QW."8YFLM01.0000.00I-1".EPL_FB_OUT_36_I2008_S25Out;
	Cyclic#1.::gFB.Out.Array[37] AT %QW."8YFLM01.0000.00I-1".EPL_FB_OUT_37_I2008_S26Out;
	Cyclic#1.::gFB.Out.Array[38] AT %QW."8YFLM01.0000.00I-1".EPL_FB_OUT_38_I2008_S27Out;
	Cyclic#1.::gFB.Out.Array[39] AT %QW."8YFLM01.0000.00I-1".EPL_FB_OUT_39_I2008_S28Out;
	Cyclic#1.::gFB.Out.Array[4] AT %QW."8YFLM01.0000.00I-1".EPL_FB_OUT_4_I2008_S05Out;
	Cyclic#1.::gFB.Out.Array[40] AT %QW."8YFLM01.0000.00I-1".EPL_FB_OUT_40_I2008_S29Out;
	Cyclic#1.::gFB.Out.Array[41] AT %QW."8YFLM01.0000.00I-1".EPL_FB_OUT_41_I2008_S2AOut;
	Cyclic#1.::gFB.Out.Array[42] AT %QW."8YFLM01.0000.00I-1".EPL_FB_OUT_42_I2008_S2BOut;
	Cyclic#1.::gFB.Out.Array[43] AT %QW."8YFLM01.0000.00I-1".EPL_FB_OUT_43_I2008_S2COut;
	Cyclic#1.::gFB.Out.Array[44] AT %QW."8YFLM01.0000.00I-1".EPL_FB_OUT_44_I2008_S2DOut;
	Cyclic#1.::gFB.Out.Array[45] AT %QW."8YFLM01.0000.00I-1".EPL_FB_OUT_45_I2008_S2EOut;
	Cyclic#1.::gFB.Out.Array[46] AT %QW."8YFLM01.0000.00I-1".EPL_FB_OUT_46_I2008_S2FOut;
	Cyclic#1.::gFB.Out.Array[47] AT %QW."8YFLM01.0000.00I-1".EPL_FB_OUT_47_I2008_S30Out;
	Cyclic#1.::gFB.Out.Array[48] AT %QW."8YFLM01.0000.00I-1".EPL_FB_OUT_48_I2008_S31Out;
	Cyclic#1.::gFB.Out.Array[49] AT %QW."8YFLM01.0000.00I-1".EPL_FB_OUT_49_I2008_S32Out;
	Cyclic#1.::gFB.Out.Array[5] AT %QW."8YFLM01.0000.00I-1".EPL_FB_OUT_5_I2008_S06Out;
	Cyclic#1.::gFB.Out.Array[50] AT %QW."8YFLM01.0000.00I-1".EPL_FB_OUT_50_I2008_S33Out;
	Cyclic#1.::gFB.Out.Array[51] AT %QW."8YFLM01.0000.00I-1".EPL_FB_OUT_51_I2008_S34Out;
	Cyclic#1.::gFB.Out.Array[52] AT %QW."8YFLM01.0000.00I-1".EPL_FB_OUT_52_I2008_S35Out;
	Cyclic#1.::gFB.Out.Array[53] AT %QW."8YFLM01.0000.00I-1".EPL_FB_OUT_53_I2008_S36Out;
	Cyclic#1.::gFB.Out.Array[54] AT %QW."8YFLM01.0000.00I-1".EPL_FB_OUT_54_I2008_S37Out;
	Cyclic#1.::gFB.Out.Array[55] AT %QW."8YFLM01.0000.00I-1".EPL_FB_OUT_55_I2008_S38Out;
	Cyclic#1.::gFB.Out.Array[56] AT %QW."8YFLM01.0000.00I-1".EPL_FB_OUT_56_I2008_S39Out;
	Cyclic#1.::gFB.Out.Array[57] AT %QW."8YFLM01.0000.00I-1".EPL_FB_OUT_57_I2008_S3AOut;
	Cyclic#1.::gFB.Out.Array[58] AT %QW."8YFLM01.0000.00I-1".EPL_FB_OUT_58_I2008_S3BOut;
	Cyclic#1.::gFB.Out.Array[59] AT %QW."8YFLM01.0000.00I-1".EPL_FB_OUT_59_I2008_S3COut;
	Cyclic#1.::gFB.Out.Array[6] AT %QW."8YFLM01.0000.00I-1".EPL_FB_OUT_6_I2008_S07Out;
	Cyclic#1.::gFB.Out.Array[60] AT %QW."8YFLM01.0000.00I-1".EPL_FB_OUT_60_I2008_S3DOut;
	Cyclic#1.::gFB.Out.Array[61] AT %QW."8YFLM01.0000.00I-1".EPL_FB_OUT_61_I2008_S3EOut;
	Cyclic#1.::gFB.Out.Array[62] AT %QW."8YFLM01.0000.00I-1".EPL_FB_OUT_62_I2008_S3FOut;
	Cyclic#1.::gFB.Out.Array[63] AT %QW."8YFLM01.0000.00I-1".EPL_FB_OUT_63_I2008_S40Out;
	Cyclic#1.::gFB.Out.Array[64] AT %QW."8YFLM01.0000.00I-1".EPL_FB_OUT_64_I2008_S41Out;
	Cyclic#1.::gFB.Out.Array[65] AT %QW."8YFLM01.0000.00I-1".EPL_FB_OUT_65_I2008_S42Out;
	Cyclic#1.::gFB.Out.Array[66] AT %QW."8YFLM01.0000.00I-1".EPL_FB_OUT_66_I2008_S43Out;
	Cyclic#1.::gFB.Out.Array[67] AT %QW."8YFLM01.0000.00I-1".EPL_FB_OUT_67_I2008_S44Out;
	Cyclic#1.::gFB.Out.Array[68] AT %QW."8YFLM01.0000.00I-1".EPL_FB_OUT_68_I2008_S45Out;
	Cyclic#1.::gFB.Out.Array[69] AT %QW."8YFLM01.0000.00I-1".EPL_FB_OUT_69_I2008_S46Out;
	Cyclic#1.::gFB.Out.Array[7] AT %QW."8YFLM01.0000.00I-1".EPL_FB_OUT_7_I2008_S08Out;
	Cyclic#1.::gFB.Out.Array[70] AT %QW."8YFLM01.0000.00I-1".EPL_FB_OUT_70_I2008_S47Out;
	Cyclic#1.::gFB.Out.Array[71] AT %QW."8YFLM01.0000.00I-1".EPL_FB_OUT_71_I2008_S48Out;
	Cyclic#1.::gFB.Out.Array[72] AT %QW."8YFLM01.0000.00I-1".EPL_FB_OUT_72_I2008_S49Out;
	Cyclic#1.::gFB.Out.Array[73] AT %QW."8YFLM01.0000.00I-1".EPL_FB_OUT_73_I2008_S4AOut;
	Cyclic#1.::gFB.Out.Array[74] AT %QW."8YFLM01.0000.00I-1".EPL_FB_OUT_74_I2008_S4BOut;
	Cyclic#1.::gFB.Out.Array[75] AT %QW."8YFLM01.0000.00I-1".EPL_FB_OUT_75_I2008_S4COut;
	Cyclic#1.::gFB.Out.Array[76] AT %QW."8YFLM01.0000.00I-1".EPL_FB_OUT_76_I2008_S4DOut;
	Cyclic#1.::gFB.Out.Array[77] AT %QW."8YFLM01.0000.00I-1".EPL_FB_OUT_77_I2008_S4EOut;
	Cyclic#1.::gFB.Out.Array[78] AT %QW."8YFLM01.0000.00I-1".EPL_FB_OUT_78_I2008_S4FOut;
	Cyclic#1.::gFB.Out.Array[79] AT %QW."8YFLM01.0000.00I-1".EPL_FB_OUT_79_I2008_S50Out;
	Cyclic#1.::gFB.Out.Array[8] AT %QW."8YFLM01.0000.00I-1".EPL_FB_OUT_8_I2008_S09Out;
	Cyclic#1.::gFB.Out.Array[80] AT %QW."8YFLM01.0000.00I-1".EPL_FB_OUT_80_I2008_S51Out;
	Cyclic#1.::gFB.Out.Array[81] AT %QW."8YFLM01.0000.00I-1".EPL_FB_OUT_81_I2008_S52Out;
	Cyclic#1.::gFB.Out.Array[82] AT %QW."8YFLM01.0000.00I-1".EPL_FB_OUT_82_I2008_S53Out;
	Cyclic#1.::gFB.Out.Array[83] AT %QW."8YFLM01.0000.00I-1".EPL_FB_OUT_83_I2008_S54Out;
	Cyclic#1.::gFB.Out.Array[84] AT %QW."8YFLM01.0000.00I-1".EPL_FB_OUT_84_I2008_S55Out;
	Cyclic#1.::gFB.Out.Array[85] AT %QW."8YFLM01.0000.00I-1".EPL_FB_OUT_85_I2008_S56Out;
	Cyclic#1.::gFB.Out.Array[86] AT %QW."8YFLM01.0000.00I-1".EPL_FB_OUT_86_I2008_S57Out;
	Cyclic#1.::gFB.Out.Array[87] AT %QW."8YFLM01.0000.00I-1".EPL_FB_OUT_87_I2008_S58Out;
	Cyclic#1.::gFB.Out.Array[88] AT %QW."8YFLM01.0000.00I-1".EPL_FB_OUT_88_I2008_S59Out;
	Cyclic#1.::gFB.Out.Array[89] AT %QW."8YFLM01.0000.00I-1".EPL_FB_OUT_89_I2008_S5AOut;
	Cyclic#1.::gFB.Out.Array[9] AT %QW."8YFLM01.0000.00I-1".EPL_FB_OUT_9_I2008_S0AOut;
	Cyclic#1.::gFB.Out.Array[90] AT %QW."8YFLM01.0000.00I-1".EPL_FB_OUT_90_I2008_S5BOut;
	Cyclic#1.::gFB.Out.Array[91] AT %QW."8YFLM01.0000.00I-1".EPL_FB_OUT_91_I2008_S5COut;
	Cyclic#1.::gFB.Out.Array[92] AT %QW."8YFLM01.0000.00I-1".EPL_FB_OUT_92_I2008_S5DOut;
	Cyclic#1.::gFB.Out.Array[93] AT %QW."8YFLM01.0000.00I-1".EPL_FB_OUT_93_I2008_S5EOut;
	Cyclic#1.::gFB.Out.Array[94] AT %QW."8YFLM01.0000.00I-1".EPL_FB_OUT_94_I2008_S5FOut;
	Cyclic#1.::gFB.Out.Array[95] AT %QW."8YFLM01.0000.00I-1".EPL_FB_OUT_95_I2008_S60Out;
	Cyclic#1.::gFB.Out.Array[96] AT %QW."8YFLM01.0000.00I-1".EPL_FB_OUT_96_I2008_S61Out;
	Cyclic#1.::gFB.Out.Array[97] AT %QW."8YFLM01.0000.00I-1".EPL_FB_OUT_97_I2008_S62Out;
	Cyclic#1.::gFB.Out.Array[98] AT %QW."8YFLM01.0000.00I-1".EPL_FB_OUT_98_I2008_S63Out;
	Cyclic#1.::gFB.Out.Array[99] AT %QW."8YFLM01.0000.00I-1".EPL_FB_OUT_99_I2008_S64Out;
END_VAR
```

### AssemConf.assembly6d - 4PPC70_0573_20B/mapp6D/AssemConf.assembly6d
```
Element g6dAssembly (Type=assembly6d)
  Simulation6D = SimOn
  Shuttles:
    MaxShuttleCount = 2
    ShuttleIDMode = RealTimeID
    DefaultPosition:
      DefZ = 1.0
      DefRx = 0
      DefRy = 0
      DefRz = 0
    Limits:
      InPlaneLimits:
        InPlaneVelLim = 1.0
        InPlaneAccLim = 10.0
        InPlaneEmergDec = 10.0
      ShortAxLim:
        ShortAxAccLim:
          AccZLim = 10.0
          AccRxLim = 10.0
          AccRyLim = 10.0
          AccRzLim = 10.0
        ShortAxVelLim:
          VelZLim = 0.15
          VelRxLim = 0.1
          VelRyLim = 0.1
          VelRzLim = 0.3
  CyclicChannel6D:
    ReadChannel:
      Xaxis = TRUE
      Yaxis = TRUE
      Zaxis = TRUE
      Rxaxis = TRUE
      Ryaxis = TRUE
      Rzaxis = TRUE
  Fieldbus6D:
    SyncMode6D = ExternalPlkSync
    NodeNumber = 101
  IOMapp:
    Input = ::gFB.In
    Output = ::gFB.Out
  Layout:
    Layout6D[1] = Layout6D_1
  Visualization:
    MonitoringPv = ::gAssemblyMon
    VisPv
    ProcessingTaskClass = 2
```

### LayoutConf.layout6d - 4PPC70_0573_20B/mapp6D/LayoutConf.layout6d
```
Element Layout6D_1 (Type=layout6d)
  Segments:
    SegRow = 1
    SegCol = 2
    Segment[1]:
      X = 0
      Y = 0
      Name
      IsMaster = True
    Segment[2]:
      X = 1
      Y = 0
      Name
      IsMaster = False
```

## Configuration X20CP1685

CPU X20CP1685, AutomationRuntime B4.91, Build 6.3.0, Safety 0.0, Vc V4.72.2

### Task classes (Cpu.sw)
```
Cyclic#1 (cycle 2000 us, tolerance 0 us):
  Acp6DCtrl <- Source.Core.Acp6DCtrl.prg
  ConvSyncDe <- (binary)
  WaveDemo <- (binary)
  ConvUnload <- (binary)
  KalmanTes1 <- (binary)
  VariedMovD <- (binary)
  MacroDemo <- (binary)
  KalmanTest <- (binary)
  RoutingDem <- (binary)
  ProcSt2 <- (binary)
  ProcSt1 <- (binary)
  CycChlCfg <- (binary)
  InspectSt <- (binary)
  DofDemo <- (binary)
  ProcessDem <- (binary)
  DanceDemoC <- (binary)
Cyclic#2 (cycle 4000 us, tolerance 4000 us):
  Program <- Source.Core.Program.prg
  RoutingDef <- Source.Core.RoutingDefinitions.prg
  PipetteSta <- Source.Core.PipetteStations.prg
  Stations <- Source.Core.Stations.prg
  DyeTipStat <- Source.Core.DyeTipStations.prg
Cyclic#4 (cycle 16000 us, tolerance 16000 us):
  Main <- Source.Core.Main.prg
Cyclic#8 (cycle 2000 us):
  RDICore <- Source.Core.RDICore.prg [disabled]
  BuildVer <- Source.BuildVersion.BuildVer.prg
  Vis <- Source.ScnViewer.Vis.prg
DataObjects: McAcpSys
NcDataObjects: mcdrivelog, AcpParTab
Binaries: FWRules, mvLoader, udbdef, TCLang, TCData, arcoal, arsvcreg, arflatprv, iomap, asfw, Role, ashwd, sysconf, arconfig, ashwac, User, TC, AssemConf, LayoutConf, mCoWebSc, CockpitSet, mcacpdrv, McAcpSim, McProfGen, McMechSys, MotConf, Hierarchy, VaxisConf, GroupConf, MechConf, FeatConf, AxisConf, FileConf, RecConf, Config_1, Config_2, OpcUaSrv, Config, Settings, CfgRecipe, CITT_FileU, CITT_Alarm, CITT_Recip, Config_4, Config_5, Config_3, Config_6, Config_8, Config_9, Config_7, Config_10, TraceConfi
Libraries: Acp6dHlpr, McBase, McAcp6D, AsSem, ArEventLog, runtime, Router6D, StnLogic, arssl, fileio, standard, astime, asieccon, asbrstr, mpbase, sys_lib, dataobj, asmem, asio, asarprof, powerlnk, asepl, asarlog, aruser, McAcpTrak, MpAxis
```

### Hardware
```
8YFLM01.0000.00I-1 : 8YFLM01.0000.00I-1 v0.0.0.1  [PLK1 -> X20CP1685.IF3 (NodeNumber=101) [Cable Type=PowerlinkCable, Length=10, Version=1.0.0.3]]
  Supervision = off
X20CP1685 : X20CP1685 v1.4.0.0
  Connector IF2:
    ActivateDevice = 1
    Mode = Manual
    InternetAddress = 192.168.10.81
    SubnetMask = 255.255.255.0
    ActivateSnmp = 2
  Connector IF3:
    CycleTime = 1000
  ConfigurationID = OnsiteDemo_C80
  TimerDeviceType = EPLX2X
  TimerDevice = X20CP1685.IF3
  TaskClassIdleTime = 2000
  Cyclic1Duration = 2000
  Cyclic1Tolerance = 0
  Cyclic2Duration = 4000
  Cyclic2Tolerance = 4000
  Cyclic3Duration = 8000
  Cyclic3Tolerance = 8000
  Cyclic4Duration = 16000
  Cyclic4Tolerance = 16000
  Cyclic5Duration = 32000
  Cyclic5Tolerance = 32000
  Cyclic6Duration = 64000
  Cyclic6Tolerance = 64000
  Cyclic7Duration = 128000
  Cyclic7Tolerance = 128000
  Cyclic8Duration = 2000
  FileDevice1
  FileDeviceName1 = 6DMacro
  FileDevicePath1 = F:\Macros
  FileDevice2
  FileDeviceName2 = CNC_PrgDir
  FileDevicePath2 = F:/Programs/
  FileDevice3
  FileDeviceName3 = Recipe
  FileDevicePath3 = F:/Recipes/
  FileDevice4
  FileDeviceName4 = TeachFileDev
  FileDevicePath4 = F:/Teach/
  FileDevice5
  FileDeviceName5 = SvMovies
  FileDevicePath5 = F:/SvMovie
  FileDevice6
  FileDeviceName6 = User
  FileDevicePath6 = F:\
  FileDevice7
  FileDeviceName7 = 6DData
  FileDevicePath7 = C:\
  FtpUser1
  FtpUsername1 = bur  // user
  FtpUserPassword1 = kzPdX7T05qFX/2O0oq22KZRISpE2rDw4PeEeBt2Wff8=  // user
  FtpUserSalt1 = NaiTqhR1
  FTPAccessRight1 = 0
  FTPdevice1 = ALL
  ActivateOpcUa = 1
  OpcUaInformationModels_PV_Version = 1
```

### AssemConf.assembly6d - X20CP1685/mapp6D/AssemConf.assembly6d
```
Element g6dAssembly (Type=assembly6d)
  Simulation6D = SimOn
  Shuttles:
    MaxShuttleCount = 5
    ShuttleIDMode = RealTimeID
    DefaultPosition:
      DefZ = 1.0
      DefRx = 0
      DefRy = 0
      DefRz = 0
    Limits:
      InPlaneLimits:
        InPlaneVelLim = 1.0
        InPlaneAccLim = 10.0
        InPlaneEmergDec = 10.0
      ShortAxLim:
        ShortAxAccLim:
          AccZLim = 10.0
          AccRxLim = 10.0
          AccRyLim = 10.0
          AccRzLim = 10.0
        ShortAxVelLim:
          VelZLim = 0.15
          VelRxLim = 0.1
          VelRyLim = 0.1
          VelRzLim = 0.3
  CyclicChannel6D:
    ReadChannel:
      Xaxis = TRUE
      Yaxis = TRUE
      Zaxis = TRUE
      Rxaxis = TRUE
      Ryaxis = TRUE
      Rzaxis = TRUE
  Fieldbus6D:
    SyncMode6D = ExternalPlkSync
    NodeNumber = 101
  IOMapp:
    Input = ::gFB.In
    Output = ::gFB.Out
  Layout:
    Layout6D[1] = Layout6D_1
  Visualization:
    MonitoringPv
    VisPv
    ProcessingTaskClass = 4
```

### LayoutConf.layout6d - X20CP1685/mapp6D/LayoutConf.layout6d
```
Element Layout6D_1 (Type=layout6d)
  Segments:
    SegRow = 3
    SegCol = 3
    Segment[1]:
      X = 0
      Y = 0
      Name
      IsMaster = True
    Segment[2]:
      X = 0
      Y = 1
      Name
      IsMaster = False
    Segment[3]:
      X = 0
      Y = 2
      Name
      IsMaster = False
    Segment[4]:
      X = 1
      Y = 0
      Name
      IsMaster = False
    Segment[5]:
      X = 1
      Y = 1
      Name
      IsMaster = False
    Segment[6]:
      X = 1
      Y = 2
      Name
      IsMaster = False
    Segment[7]:
      X = 2
      Y = 1
      Name
      IsMaster = False
```

## Logical view

Binary libraries used (declarations not repeated): operator, runtime, astime, AsIecCon, AsZip, FileIO, standard, AsBrStr, sys_lib, brsystem, MpFile, MpBase, CoTrace, MpRecipe, AsSem, ArEventLog, McBase 5.17.9, McAcp6D 1.01.9

### Global.typ - Global data types
```iecst
TYPE
	gFBType : 	STRUCT  (*6D Interfaces*)
		In : Mc6DControllerFBIOType; (*Inputs*)
		Out : Mc6DControllerFBIOType; (*Outputs*)
	END_STRUCT;
END_TYPE

(************************* Main If Typ*)

TYPE
	MainIfTyp : 	STRUCT
		Cmd : MainIfCmdTyp;
		Par : USINT;
		Sts : USINT;
	END_STRUCT;
	MainIfCmdTyp : 	STRUCT
		Power : BOOL;
		Run : BOOL;
		ErrorReset : BOOL;
	END_STRUCT;
	SystemRecipeIfTyp : 	STRUCT
		DefaultVel : REAL;
		DefaultAccel : REAL;
		DefaultWaitTime : UDINT;
		StartupPars : StartupPars;
		WellRecipe : ARRAY[0..1]OF FillRecipeTyp;
		PipettePars : PipettePars;
	END_STRUCT;
	StartupPars : 	STRUCT
		MoveAsyncPars : McAcp6DMoveInPlaneAsyncParType;
	END_STRUCT;
	PipettePars : 	STRUCT
		HomePosition : REAL;
		Vel : REAL;
		SampleDistance : REAL;
		WellDistance : REAL;
	END_STRUCT;
END_TYPE

(************************* Acp6D Types*)

TYPE
	Acp6DIfTyp : 	STRUCT
		Cmd : Acp6DCmdsTyp;
		Par : Acp6DParTyp;
		Sts : Acp6DStsTyp;
	END_STRUCT;
	Acp6DCmdsTyp : 	STRUCT
		Power : BOOL;
		Reset : BOOL;
		ResetInfo : BOOL;
	END_STRUCT;
	Acp6DParTyp : 	STRUCT
		ShuttleCount : USINT;
		Asm : Mc6DAssemblyType;
	END_STRUCT;
	Acp6DStsTyp : 	STRUCT
		Error : BOOL;
		AssemblyInfo : McAcp6DAsmGetInfoType;
		AssemblyDisabled : BOOL;
		AssemblyReady : BOOL;
		AssemblyHoming : BOOL;
		AssemblyStopping : BOOL;
		AssemblyStartup : BOOL;
		AssemblyErrorStop : BOOL;
	END_STRUCT;
END_TYPE

(************************** Shuttle If Types*)

TYPE
	ShuttleIfTyp : 	STRUCT
		Cmd : ShuttleIfCmdTyp;
		Par : ShuttleIfParTyp;
		Cfg : ShuttleIfCfgTyp;
		Sts : ShuttleIfStsTyp;
	END_STRUCT;
	ShuttleIfCmdTyp : 	STRUCT
		Reset : BOOL;
	END_STRUCT;
	ShuttleIfParTyp : 	STRUCT
		New_Member : USINT;
	END_STRUCT;
	ShuttleIfCfgTyp : 	STRUCT
		ID : UINT;
		Shuttle : Mc6DShuttleType;
		RouterShuttle : rl6dShuttleType;
	END_STRUCT;
	ShuttleIfStsTyp : 	STRUCT
		Available : BOOL;
		Error : BOOL;
		ErrorID : UDINT;
	END_STRUCT;
END_TYPE

(*Routing Helper Types*)

TYPE
	DestTyp : 	STRUCT
		StationName : STRING[80];
		Position : rl6dPositionType;
		Entry : DestPathTyp;
		Exit : DestPathTyp;
		RecoveryPts : rl6dPositionType;
		Destination : rl6dDestinationType;
	END_STRUCT;
	DestPathTyp : 	STRUCT
		Path : rl6dPathType;
		PathPoints : ARRAY[0..2]OF rl6dPositionType;
		Name : STRING[80];
		Length : USINT;
	END_STRUCT;
	WaypointTyp : 	STRUCT
		Position : rl6dPositionType;
		Name : STRING[80];
		Waypoint : rl6dWaypointType;
		Destinations : ARRAY[0..5]OF DestinationsEnum;
		NextWaypoint : WaypointListEnum;
	END_STRUCT;
	WaypointListEnum :
		(
		WP_NONE,
		WP_1,
		WP_2,
		WP_3,
		WP_4,
		WP_5
		);
	StationsIfTyp : 	STRUCT
		Cmd : StationsCmdTyp;
		Par : StationsParTyp;
		Sts : StationsStsTyp;
	END_STRUCT;
	StationsCmdTyp : 	STRUCT
		Enable : BOOL;
		Run : BOOL;
		Recover : BOOL;
		RequestIncubator : BOOL;
		RequestPipette : ARRAY[0..1]OF BOOL;
		RequestDye : BOOL;
		RequestTip : BOOL;
		RequestFreshShuttle : BOOL;
		RequestAnalyzer : BOOL;
	END_STRUCT;
	StationsParTyp : 	STRUCT
		Incubator : IncubatorParTyp;
		Analyzer : IncubatorParTyp;
		Pipette : ARRAY[0..1]OF PipetteParTyp;
		Dye : DyeTipParTyp;
		Tip : DyeTipParTyp;
	END_STRUCT;
	PipetteParTyp : 	STRUCT
		NextStation : DestinationsEnum;
		Waypoint : WaypointListEnum;
		ShuttleType : ShuttleType;
	END_STRUCT;
	DyeTipParTyp : 	STRUCT
		RequestDestination : DestinationsEnum;
		Waypoint : WaypointListEnum;
	END_STRUCT;
	IncubatorParTyp : 	STRUCT
		SampleType : ColorEnum;
		NextStation : DestinationsEnum;
		Waypoint : WaypointListEnum;
	END_STRUCT;
	StationsStsTyp : 	STRUCT
		RoutingInitalized : BOOL;
		IncubatorShuttlePresent : BOOL;
		IncubatorActive : BOOL;
		PipetteActive : ARRAY[0..1]OF BOOL;
		PipetteNeedSample : ARRAY[0..1]OF BOOL;
		PipetteShuttlePresent : ARRAY[0..1]OF BOOL;
		PipetteReadyForShuttle : ARRAY[0..1]OF BOOL;
		TipsShuttlePresent : BOOL;
		DyeShuttlePresent : BOOL;
		AnalyzerShuttlePresent : BOOL;
	END_STRUCT;
	AnalyzerParTyp : 	STRUCT
		NextStation : DestinationsEnum;
		Waypoint : WaypointListEnum;
		PipetteIndex : USINT;
	END_STRUCT;
END_TYPE
```

### Global.var - Global variables
```iecst
VAR
	gFB : gFBType; (*6D Interfaces*)
END_VAR
VAR CONSTANT
	NUM_SHUTTLES : USINT := 5;
	MAX_SH_IDX : USINT := NUM_SHUTTLES - 1;
END_VAR
(*********************** Interface Variables*)
VAR
	gAcp6DIf : Acp6DIfTyp;
	gSysRecipe : SystemRecipeIfTyp;
	gSystemIf : MainIfTyp;
	gShIfs : ARRAY[0..MAX_SH_IDX] OF ShuttleIfTyp;
	gStationsIf : StationsIfTyp;
END_VAR
(*Routing Variables*)
VAR
	gDests : ARRAY[0..9] OF DestTyp;
	gWps : ARRAY[0..6] OF WaypointTyp;
END_VAR
```

### Package Logical/Libraries - Global libraries

### Library Logical/Libraries/rdiAcp6D (IEC)

#### Types.typ - Exported data types
```iecst
(*Parameter structures*)

TYPE
	Pars6D_typ : 	STRUCT
		Linear : McAcp6DInPlaneParType;
		Arc : McAcp6DArcParType;
		ShortAxis : McAcp6DShortAxParType;
		Async : MoveAsync_typ;
		SixDOF : McAcp6DMove6DParType;
		Levitation : McAcp6DLevitationParType;
		Buffer : UINT;
	END_STRUCT;
	MoveAsync_typ : 	STRUCT
		Velocity : REAL;
		Acceleration : REAL;
		ShuttleTable : ARRAY[0..rdiMAX_ASYNC_SHUTTLES_M1]OF AsyncShuttle_typ;
	END_STRUCT;
	AsyncShuttle_typ : 	STRUCT
		X : REAL;
		Y : REAL;
		ShuttleID : UINT;
	END_STRUCT;
END_TYPE

(*Output structures*)

TYPE
	AsmStatus_typ : 	STRUCT
		AssemblyDisabled : BOOL;
		AssemblyReady : BOOL;
		AssemblyHoming : BOOL;
		AssemblyStopping : BOOL;
		AssemblyStartUp : BOOL;
		AssemblyErrorStop : BOOL;
	END_STRUCT;
	ShuttleInfo_typ : 	STRUCT
		Axis : Mc6DShuttleType;
		ShuttleID : UINT;
		State : McAcp6DShStateEnum;
		Position : McAcp6DShPositionType;
	END_STRUCT;
	ShuttleBufferInfo_typ : 	STRUCT
		ShuttleID : UINT;
		State : McAcp6DBufferStateEnum;
		NumberOfCommands : UINT;
	END_STRUCT;
END_TYPE

(*Internal 6D function block organization*)

TYPE
	Internal6DCore_typ : 	STRUCT
		State : Core6DState_enum;
		Status : Internal6DCoreStatus_typ;
		FB : FB6D_typ;
	END_STRUCT;
	Core6DState_enum :
		(
		rdi_VALIDATE_ASSEMBLY_REF,
		rdi_ENABLE_ASM_READ_STATUS,
		rdi_WAIT_FOR_POWER_ON,
		rdi_GET_ASM_INFO,
		rdi_VALIDATE_GET_SHUTTLES,
		rdi_GET_SHUTTLES,
		rdi_GET_SHUTTLES_NEXT,
		rdi_GET_SHUTTLE_INFO,
		rdi_CHECK_SHUTTLE_INFO,
		rdi_WAIT_FOR_COMMAND,
		rdi_MOVE_LINEAR,
		rdi_MOVE_ARC,
		rdi_MOVE_SHORT,
		rdi_MOVE_6DOF,
		rdi_MOVE_ASYNC,
		rdi_ASM_STOP,
		rdi_SHUTTLE_STOP,
		rdi_ASM_HALT,
		rdi_SHUTTLE_HALT,
		rdi_ASM_LEVITATION,
		rdi_SHUTTLE_LEVITATION,
		rdi_ASM_BUFFER,
		rdi_SHUTTLE_BUFFER,
		rd_SHUTTLE_BUFFER_STATUS,
		rdi_ASM_REBOOT,
		rdi_POWER_OFF,
		rdi_SHUTTLE_RECOVER,
		rdi_ERROR
		);
	Internal6DCoreStatus_typ : 	STRUCT
		AsmGetInfoShuttleCount : UINT;
		GetShuttleCount : USINT;
		OldShuttleID : UINT;
		SelectedShuttleAxis : Mc6DShuttleType;
	END_STRUCT;
	FB6D_typ : 	STRUCT
		Asm : AsmFB6D_typ;
		Stop : StopFB6D_typ;
		Halt : HaltFB6D_typ;
		Move : MoveFB6D_typ;
		Shuttle : ShuttleFB6D_typ;
		Levitation : LevitationFB6D_typ;
		Buffer : BufferFB6D_typ;
	END_STRUCT;
	AsmFB6D_typ : 	STRUCT
		AsmPowerOn : MC_BR_AsmPowerOn_Acp6D;
		AsmPowerOff : MC_BR_AsmPowerOff_Acp6D;
		AsmReboot : MC_BR_AsmReboot_Acp6D;
		AsmGetInfo : MC_BR_AsmGetInfo_Acp6D;
		AsmReadStatus : MC_BR_AsmReadStatus_Acp6D;
		AsmGetShuttle : MC_BR_AsmGetShuttle_Acp6D;
	END_STRUCT;
	StopFB6D_typ : 	STRUCT
		AsmStop : MC_BR_AsmStop_Acp6D;
		ShStop : MC_BR_ShStop_Acp6D;
	END_STRUCT;
	HaltFB6D_typ : 	STRUCT
		AsmHalt : MC_BR_AsmHalt_Acp6D;
		ShHalt : MC_BR_ShHalt_Acp6D;
	END_STRUCT;
	MoveFB6D_typ : 	STRUCT
		Linear : MC_BR_MoveInPlane_Acp6D;
		Arc : MC_BR_MoveArc_Acp6D;
		Short : MC_BR_MoveShortAxis_Acp6D;
		Async : MC_BR_MoveInPlaneAsync_Acp6D;
		SixDOF : MC_BR_Move6D_Acp6D;
	END_STRUCT;
	ShuttleFB6D_typ : 	STRUCT
		ShReadInfo : ARRAY[0..MAX_NUM_SHUTTLES_M1]OF MC_BR_ShReadInfo_Acp6D;
		ShRecover : MC_BR_ShRecover_Acp6D;
	END_STRUCT;
	LevitationFB6D_typ : 	STRUCT
		AsmLevitation : MC_BR_AsmLevitation_Acp6D;
		ShLevitation : MC_BR_ShLevitation_Acp6D;
	END_STRUCT;
	BufferFB6D_typ : 	STRUCT
		AsmBuffer : MC_BR_AsmBuffer_Acp6D;
		ShBuffer : MC_BR_ShBuffer_Acp6D;
	END_STRUCT;
END_TYPE
```

#### Constants.var - Exported constants
```iecst
VAR CONSTANT
	MAX_NUM_SHUTTLES : USINT := 2;
	MAX_NUM_SHUTTLES_M1 : USINT := MAX_NUM_SHUTTLES - 1;
	rdiERROR_INVALID_PAR : DINT := -1065795584;
	rdiMAX_ASYNC_SHUTTLES : USINT := 78;
	rdiMAX_ASYNC_SHUTTLES_M1 : USINT := rdiMAX_ASYNC_SHUTTLES - 1;
END_VAR
```

#### rdiAcp6D.fun - Exported functions and function blocks
```iecst
{REDUND_ERROR} FUNCTION_BLOCK rdi6DCore (*TODO: Add your comment here*) (*$GROUP=User,$CAT=User,$GROUPICON=User.png,$CATICON=User.png*)
	VAR_INPUT
		AsmRef : REFERENCE TO Mc6DAssemblyType;
		Enable : BOOL;
		ErrorReset : BOOL;
		Parameters : REFERENCE TO Pars6D_typ;
		Power : BOOL;
		AsmStop : BOOL;
		ShStop : BOOL;
		AsmHalt : BOOL;
		ShHalt : BOOL;
		AsmResume : BOOL;
		ShResume : BOOL;
		AsmLevitation : BOOL;
		ShLevitation : BOOL;
		AsmBuffer : BOOL;
		ShBuffer : BOOL;
		ShuttleID : UINT;
		Reboot : BOOL;
		MoveLinear : BOOL;
		MoveArc : BOOL;
		MoveShort : BOOL;
		MoveAsync : BOOL;
		Move6DOF : BOOL;
		ShRecover : BOOL;
	END_VAR
	VAR_OUTPUT
		Active : BOOL;
		Error : BOOL;
		ErrorID : DINT;
		PowerOn : BOOL;
		MovementActive : BOOL;
		AllShuttlesFound : BOOL;
		ValidShuttleSelected : BOOL;
		ShuttleArray : ARRAY[0..MAX_NUM_SHUTTLES_M1] OF ShuttleInfo_typ;
		AsmStatus : AsmStatus_typ;
		ShuttleBufferInfo : ShuttleBufferInfo_typ;
		CurrentState : STRING[80];
		StatusMessage : STRING[80];
	END_VAR
	VAR
		j : UINT;
		i : UINT;
		Internal : Internal6DCore_typ;
		zzEdge00000 : BOOL;
		zzEdge00001 : BOOL;
		zzEdge00002 : BOOL;
		zzEdge00003 : BOOL;
		zzEdge00004 : BOOL;
		zzEdge00005 : BOOL;
		zzEdge00006 : BOOL;
		zzEdge00007 : BOOL;
		zzEdge00008 : BOOL;
		zzEdge00009 : BOOL;
		zzEdge00010 : BOOL;
		zzEdge00011 : BOOL;
		zzEdge00012 : BOOL;
		zzEdge00013 : BOOL;
		zzEdge00014 : BOOL;
		zzEdge00015 : BOOL;
		zzEdge00016 : BOOL;
		zzEdge00017 : BOOL;
	END_VAR
END_FUNCTION_BLOCK
```

#### rdi6DCore.st
```iecst
(* TODO: Add your comment here *)
FUNCTION_BLOCK rdi6DCore

	IF Enable THEN

		CASE Internal.State OF

			rdi_VALIDATE_ASSEMBLY_REF:
				CurrentState := 'rdi_VALIDATE_ASSEMBLY_REF';

				IF AsmRef.controlif <> 0 THEN
					Internal.FB.Asm.AsmReadStatus.Assembly := ADR(AsmRef);
					Internal.FB.Asm.AsmGetInfo.Assembly := ADR(AsmRef);
					Internal.FB.Asm.AsmGetShuttle.Assembly := ADR(AsmRef);
					Internal.FB.Asm.AsmPowerOn.Assembly := ADR(AsmRef);
					Internal.FB.Asm.AsmPowerOff.Assembly := ADR(AsmRef);
					Internal.FB.Asm.AsmReboot.Assembly := ADR(AsmRef);
					Internal.FB.Move.Async.Assembly := ADR(AsmRef);
					Internal.FB.Stop.AsmStop.Assembly := ADR(AsmRef);
					Internal.FB.Halt.AsmHalt.Assembly := ADR(AsmRef);
					Internal.FB.Levitation.AsmLevitation.Assembly := ADR(AsmRef);
					Internal.FB.Buffer.AsmBuffer.Assembly := ADR(AsmRef);

					Internal.State := rdi_ENABLE_ASM_READ_STATUS;

				ELSE
					StatusMessage := 'Assembly reference not set';
				END_IF

			(* enable AsmReadStatus to get info about the system *)
			rdi_ENABLE_ASM_READ_STATUS:
				CurrentState := 'rdi_ENABLE_ASM_READ_STATUS';
				Internal.FB.Asm.AsmReadStatus.Enable := TRUE;

				IF Internal.FB.Asm.AsmReadStatus.Valid THEN
					Internal.State := rdi_WAIT_FOR_POWER_ON;
				END_IF

			(* wait for user to issue the Power command *)
			rdi_WAIT_FOR_POWER_ON:
				CurrentState := 'rdi_WAIT_FOR_POWER_ON';
				AllShuttlesFound := FALSE;
				Internal.FB.Asm.AsmPowerOn.Execute := Power;
				IF Internal.FB.Asm.AsmReadStatus.AssemblyReady THEN
					brsmemset(ADR(ShuttleArray), 0, SIZEOF(ShuttleArray));
					brsmemset(ADR(Internal.FB.Shuttle.ShReadInfo), 0, SIZEOF(Internal.FB.Shuttle.ShReadInfo));
					Internal.FB.Asm.AsmPowerOn.Execute := FALSE;
					Internal.State := rdi_GET_ASM_INFO;
				END_IF

			rdi_GET_ASM_INFO:
				CurrentState := 'rdi_GET_ASM_INFO';
				Internal.FB.Asm.AsmGetInfo.Execute := TRUE;
				IF Internal.FB.Asm.AsmGetInfo.Done THEN
					Internal.Status.AsmGetInfoShuttleCount := Internal.FB.Asm.AsmGetInfo.AssemblyInfo.NumberOfShuttles;
					Internal.FB.Asm.AsmGetInfo.Execute := FALSE;
					Internal.Status.GetShuttleCount := 0;

					Internal.State := rdi_VALIDATE_GET_SHUTTLES;
				END_IF

			(* Reattempt to get shuttles until successful; this state will not be needed when AsmGetShuttle is more reliable *)
			rdi_VALIDATE_GET_SHUTTLES:
				CurrentState := 'rdi_VALIDATE_GET_SHUTTLES';
				StatusMessage := 'Getting Shuttles';
				Internal.FB.Asm.AsmGetShuttle.Enable := TRUE;
				IF Internal.FB.Asm.AsmGetShuttle.Valid THEN
					IF Internal.FB.Asm.AsmGetShuttle.TotalCount > 0 THEN
						Internal.State := rdi_GET_SHUTTLES;
					ELSE
						Internal.FB.Asm.AsmGetShuttle.Enable := FALSE;
					END_IF
				END_IF

			(* get the shuttles on the system and store them into a shuttle array *)
			rdi_GET_SHUTTLES:
				CurrentState := 'rdi_GET_SHUTTLES';
				Internal.FB.Asm.AsmGetShuttle.Enable := TRUE;
				IF Internal.FB.Asm.AsmGetShuttle.Valid THEN
					IF Internal.FB.Asm.AsmGetShuttle.Shuttle.controlif <> 0 THEN
						ShuttleArray[Internal.Status.GetShuttleCount].Axis := Internal.FB.Asm.AsmGetShuttle.Shuttle;
						ShuttleArray[Internal.Status.GetShuttleCount].ShuttleID := Internal.FB.Asm.AsmGetShuttle.AdditionalInfo.ShuttleID;
					END_IF

					IF Internal.FB.Asm.AsmGetShuttle.RemainingCount > 0 THEN
						Internal.FB.Asm.AsmGetShuttle.Next := TRUE;
						Internal.State := rdi_GET_SHUTTLES_NEXT;
					ELSE
						AllShuttlesFound := TRUE;
						ShuttleID := ShuttleArray[Internal.Status.GetShuttleCount].ShuttleID;
						Internal.FB.Asm.AsmGetShuttle.Enable := FALSE;
						Internal.State := rdi_GET_SHUTTLE_INFO;
					END_IF
				END_IF

			rdi_GET_SHUTTLES_NEXT:
				CurrentState := 'rdi_GET_SHUTTLES_NEXT';
				Internal.FB.Asm.AsmGetShuttle.Next := FALSE;
				Internal.Status.GetShuttleCount := Internal.Status.GetShuttleCount + 1;
				Internal.State := rdi_GET_SHUTTLES;

			(* enable ShReadInfo for all shuttles *)
			rdi_GET_SHUTTLE_INFO:
				CurrentState := 'rdi_GET_SHUTTLE_INFO';

				FOR i := 0 TO MAX_NUM_SHUTTLES_M1 DO
					IF ShuttleArray[i].Axis.controlif <> 0 THEN
						Internal.FB.Shuttle.ShReadInfo[i].Shuttle := ADR(ShuttleArray[i].Axis);
						Internal.FB.Shuttle.ShReadInfo[i].Enable := TRUE;
					END_IF
				END_FOR

				Internal.State := rdi_CHECK_SHUTTLE_INFO;

			rdi_CHECK_SHUTTLE_INFO:
				(* I found that if you remove a shuttle, power off the controller, and power on again, the controller will
					still see the removed shuttle. So if the shuttle is in the RESERVED state right after power on, something
					is probably wrong and the shuttle should be deleted. If not, since the non-existing shuttle axis is still valid,
					things can get hung up *)

				FOR i := 0 TO MAX_NUM_SHUTTLES_M1 DO
					IF Internal.FB.Shuttle.ShReadInfo[i].ShuttleInfo.State = mcACP6D_SH_STATE_RESERVED THEN
						brsmemset(ADR(ShuttleArray[i]), 0, SIZEOF(ShuttleArray[i]));
						brsmemset(ADR(Internal.FB.Shuttle.ShReadInfo[i]), 0, SIZEOF(Internal.FB.Shuttle.ShReadInfo[i]));
					END_IF
				END_FOR

				Internal.State := rdi_WAIT_FOR_COMMAND;

			(* main waiting state *)
			rdi_WAIT_FOR_COMMAND:
				CurrentState := 'rdi_WAIT_FOR_COMMAND';

				IF NOT Power THEN
					StatusMessage := 'Powering Off';
					Internal.State := rdi_POWER_OFF;
				ELSIF EDGEPOS(AsmStop) THEN
					StatusMessage := 'Stopping Assembly';
					Internal.State := rdi_ASM_STOP;
				ELSIF EDGEPOS(ShStop) AND ValidShuttleSelected THEN
					StatusMessage := 'Stopping Shuttle';
					Internal.State := rdi_SHUTTLE_STOP;
				ELSIF EDGEPOS(AsmHalt) THEN
					StatusMessage := 'Halting Assembly';
					Internal.FB.Halt.AsmHalt.Option := mcACP6D_HALT;
					Internal.State := rdi_ASM_HALT;
				ELSIF EDGEPOS(ShHalt) AND ValidShuttleSelected THEN
					StatusMessage := 'Halting Shuttle';
					Internal.FB.Halt.ShHalt.Option := mcACP6D_HALT;
					Internal.State := rdi_SHUTTLE_HALT;
				ELSIF EDGEPOS(AsmResume) THEN
					StatusMessage := 'Resuming Assembly';
					Internal.FB.Halt.AsmHalt.Option := mcACP6D_CONTINUE;
					Internal.State := rdi_ASM_HALT;
				ELSIF EDGEPOS(ShResume) AND ValidShuttleSelected THEN
					StatusMessage := 'Resuming Shuttle';
					Internal.FB.Halt.ShHalt.Option := mcACP6D_CONTINUE;
					Internal.State := rdi_SHUTTLE_HALT;
				ELSIF EDGEPOS(MoveLinear) AND ValidShuttleSelected THEN
					StatusMessage := 'Started Movement: Linear';
					Internal.State := rdi_MOVE_LINEAR;
				ELSIF EDGEPOS(MoveArc) AND ValidShuttleSelected THEN
					StatusMessage := 'Started Movement: Arc';
					Internal.State := rdi_MOVE_ARC;
				ELSIF EDGEPOS(MoveShort) AND ValidShuttleSelected THEN
					StatusMessage := 'Started Movement: Short';
					Internal.State := rdi_MOVE_SHORT;
				ELSIF EDGEPOS(Move6DOF) AND ValidShuttleSelected THEN
					StatusMessage := 'Started Movement: 6DOF';
					Internal.State := rdi_MOVE_6DOF;
				ELSIF EDGEPOS(MoveAsync) THEN
					StatusMessage := 'Started Movement: Async';
					Internal.State := rdi_MOVE_ASYNC;
				ELSIF EDGEPOS(AsmLevitation) THEN
					StatusMessage := 'Started Asm Levitation Command';
					Internal.State := rdi_ASM_LEVITATION;
				ELSIF EDGEPOS(ShLevitation) THEN
					StatusMessage := 'Started Sh Levitation Command';
					Internal.State := rdi_SHUTTLE_LEVITATION;
				ELSIF EDGEPOS(AsmBuffer) AND ValidShuttleSelected THEN
					StatusMessage := 'Started Asm Buffer Command';
					Internal.State := rdi_ASM_BUFFER;
				ELSIF EDGEPOS(ShBuffer) AND ValidShuttleSelected THEN
					StatusMessage := 'Started Sh Buffer Command';
					Internal.State := rdi_SHUTTLE_BUFFER;
				ELSIF EDGEPOS(Reboot) THEN
					StatusMessage := 'Rebooting 6D Controller';
					Internal.State := rdi_ASM_REBOOT;
				ELSIF EDGEPOS(ShRecover) THEN
					StatusMessage := 'Recovering Shuttle';
					Internal.State := rdi_SHUTTLE_RECOVER;
				END_IF

				(* check if selected shuttle changed, then check if new ID exists *)
				IF ShuttleID <> Internal.Status.OldShuttleID THEN
					FOR i := 0 TO MAX_NUM_SHUTTLES_M1 DO
						IF ShuttleID = ShuttleArray[i].ShuttleID THEN
							Internal.Status.SelectedShuttleAxis := ShuttleArray[i].Axis;
							Internal.Status.OldShuttleID := ShuttleID;
							ValidShuttleSelected := TRUE;
							EXIT;
						END_IF
					END_FOR
					IF i = MAX_NUM_SHUTTLES THEN
						Internal.Status.OldShuttleID := ShuttleID;
						ValidShuttleSelected := FALSE;
					END_IF
				END_IF

			rdi_MOVE_LINEAR:
				CurrentState := 'rdi_MOVE_LINEAR';

				Internal.FB.Move.Linear.Shuttle := ADR(Internal.Status.SelectedShuttleAxis);
				brsmemcpy(ADR(Internal.FB.Move.Linear.Parameters), ADR(Parameters.Linear), SIZEOF(McAcp6DInPlaneParType));
				Internal.FB.Move.Linear.Execute := TRUE;

				IF Internal.FB.Move.Linear.Error THEN
					Internal.FB.Move.Linear.Execute := FALSE;
					IF Internal.FB.Move.Linear.ErrorID = rdiERROR_INVALID_PAR THEN
						StatusMessage := 'Movement Linear: Invalid parameters';
						Internal.State := rdi_WAIT_FOR_COMMAND;
					ELSE
						ErrorID := Internal.FB.Move.Linear.ErrorID;
						Internal.State := rdi_ERROR;
					END_IF
				ELSIF Internal.FB.Move.Linear.Acknowledge THEN
					Internal.FB.Move.Linear.Execute := FALSE;
					Internal.State := rdi_WAIT_FOR_COMMAND;
				END_IF

			rdi_MOVE_ARC:
				CurrentState := 'rdi_MOVE_ARC';

				Internal.FB.Move.Arc.Shuttle := ADR(Internal.Status.SelectedShuttleAxis);
				brsmemcpy(ADR(Internal.FB.Move.Arc.Parameters), ADR(Parameters.Arc), SIZEOF(McAcp6DArcParType));
				Internal.FB.Move.Arc.Execute := TRUE;

				IF Internal.FB.Move.Arc.Error THEN
					Internal.FB.Move.Arc.Execute := FALSE;
					IF Internal.FB.Move.Arc.ErrorID = rdiERROR_INVALID_PAR THEN
						StatusMessage := 'Movement Arc: Invalid parameters';
						Internal.State := rdi_WAIT_FOR_COMMAND;
					ELSE

						ErrorID := Internal.FB.Move.Arc.ErrorID;
						Internal.State := rdi_ERROR;
					END_IF
				ELSIF Internal.FB.Move.Arc.Acknowledge THEN
					Internal.FB.Move.Arc.Execute := FALSE;
					Internal.State := rdi_WAIT_FOR_COMMAND;
				END_IF

			rdi_MOVE_SHORT:
				CurrentState := 'rdi_MOVE_SHORT';

				Internal.FB.Move.Short.Shuttle := ADR(Internal.Status.SelectedShuttleAxis);
				brsmemcpy(ADR(Internal.FB.Move.Short.Parameters), ADR(Parameters.ShortAxis), SIZEOF(McAcp6DShortAxParType));
				Internal.FB.Move.Short.Execute := TRUE;

				IF Internal.FB.Move.Short.Error THEN
					Internal.FB.Move.Short.Execute := FALSE;
					IF Internal.FB.Move.Short.ErrorID = rdiERROR_INVALID_PAR THEN
						StatusMessage := 'Movement Short: Invalid parameters';
						Internal.State := rdi_WAIT_FOR_COMMAND;
					ELSE
						ErrorID := Internal.FB.Move.Short.ErrorID;
						Internal.State := rdi_ERROR;
					END_IF
				ELSIF Internal.FB.Move.Short.Acknowledge THEN
					Internal.FB.Move.Short.Execute := FALSE;
					Internal.State := rdi_WAIT_FOR_COMMAND;
				END_IF

			rdi_MOVE_6DOF:
				CurrentState := 'rdi_MOVE_6DOF';

				Internal.FB.Move.SixDOF.Shuttle := ADR(Internal.Status.SelectedShuttleAxis);
				brsmemcpy(ADR(Internal.FB.Move.SixDOF.Parameters), ADR(Parameters.SixDOF), SIZEOF(McAcp6DMove6DParType));
				Internal.FB.Move.SixDOF.Execute := TRUE;

				IF Internal.FB.Move.SixDOF.Error THEN
					Internal.FB.Move.SixDOF.Execute := FALSE;
					IF Internal.FB.Move.SixDOF.ErrorID = rdiERROR_INVALID_PAR THEN
						StatusMessage := 'Movement 6DOF: Invalid parameters';
						Internal.State := rdi_WAIT_FOR_COMMAND;
					ELSE
						ErrorID := Internal.FB.Move.SixDOF.ErrorID;
						Internal.State := rdi_ERROR;
					END_IF
				ELSIF Internal.FB.Move.SixDOF.Acknowledge THEN
					Internal.FB.Move.SixDOF.Execute := FALSE;
					Internal.State := rdi_WAIT_FOR_COMMAND;
				END_IF

			rdi_MOVE_ASYNC:
				CurrentState := 'rdi_MOVE_ASYNC';
				Internal.FB.Move.Async.Execute := TRUE;

				Internal.FB.Move.Async.Parameters.Acceleration := Parameters.Async.Acceleration;
				Internal.FB.Move.Async.Parameters.Velocity := Parameters.Async.Velocity;

				FOR i := 0 TO rdiMAX_ASYNC_SHUTTLES_M1 DO
					FOR j := 0 TO MAX_NUM_SHUTTLES_M1 DO
						IF Parameters.Async.ShuttleTable[i].ShuttleID = 0 THEN
							EXIT;
						ELSIF Parameters.Async.ShuttleTable[i].ShuttleID = ShuttleArray[j].ShuttleID THEN
							Internal.FB.Move.Async.Parameters.AsyncPar[i].Shuttle := ADR(ShuttleArray[j].Axis);
							Internal.FB.Move.Async.Parameters.AsyncPar[i].X := Parameters.Async.ShuttleTable[i].X;
							Internal.FB.Move.Async.Parameters.AsyncPar[i].Y := Parameters.Async.ShuttleTable[i].Y;
							EXIT;
						END_IF
					END_FOR
					IF j = MAX_NUM_SHUTTLES THEN
						Internal.FB.Move.Async.Execute := FALSE;
						StatusMessage := 'Movement Async: Invalid Shuttle ID';
						Internal.State := rdi_WAIT_FOR_COMMAND;
						EXIT;
					END_IF
				END_FOR

				IF Internal.FB.Move.Async.Error THEN
					Internal.FB.Move.Async.Execute := FALSE;
					IF Internal.FB.Move.Async.ErrorID = rdiERROR_INVALID_PAR THEN
						StatusMessage := 'Movement Async: Invalid parameters';
						Internal.State := rdi_WAIT_FOR_COMMAND;
					ELSE
						ErrorID := Internal.FB.Move.Async.ErrorID;
						Internal.State := rdi_ERROR;
					END_IF
				ELSIF Internal.FB.Move.Async.Acknowledge THEN
					Internal.FB.Move.Async.Execute := FALSE;
					Internal.State := rdi_WAIT_FOR_COMMAND;
				END_IF

			rdi_ASM_STOP:
				CurrentState := 'rdi_ASM_STOP';
				Internal.FB.Stop.AsmStop.Execute := TRUE;

				IF Internal.FB.Stop.AsmStop.Error THEN
					Internal.FB.Stop.AsmStop.Execute := FALSE;
					ErrorID := Internal.FB.Stop.AsmStop.ErrorID;
					Internal.State := rdi_ERROR;
				ELSIF Internal.FB.Stop.AsmStop.Done THEN
					Internal.FB.Stop.AsmStop.Execute := FALSE;
					Internal.State := rdi_WAIT_FOR_COMMAND;
				END_IF

			rdi_SHUTTLE_STOP:
				CurrentState := 'rdi_SHUTTLE_STOP';
				Internal.FB.Stop.ShStop.Shuttle := ADR(Internal.Status.SelectedShuttleAxis);
				Internal.FB.Stop.ShStop.Execute := TRUE;

				IF Internal.FB.Stop.ShStop.Error THEN
					Internal.FB.Stop.ShStop.Execute := FALSE;
					ErrorID := Internal.FB.Stop.ShStop.ErrorID;
					Internal.State := rdi_ERROR;
				ELSIF Internal.FB.Stop.ShStop.Done THEN
					Internal.FB.Stop.ShStop.Execute := FALSE;
					Internal.State := rdi_WAIT_FOR_COMMAND;
				END_IF

			rdi_ASM_HALT:
				CurrentState := 'rdi_ASM_HALT';
				Internal.FB.Halt.AsmHalt.Execute := TRUE;
				//Internal.FB.Halt.AsmHalt.Option

				IF Internal.FB.Halt.AsmHalt.Error THEN
					Internal.FB.Halt.AsmHalt.Execute := FALSE;
					ErrorID := Internal.FB.Halt.AsmHalt.ErrorID;
					Internal.State := rdi_ERROR;
				ELSIF Internal.FB.Halt.AsmHalt.Done THEN
					Internal.FB.Halt.AsmHalt.Execute := FALSE;
					Internal.State := rdi_WAIT_FOR_COMMAND;
				END_IF

			rdi_SHUTTLE_HALT:
				CurrentState := 'rdi_SHUTTLE_HALT';
				Internal.FB.Halt.ShHalt.Shuttle := ADR(Internal.Status.SelectedShuttleAxis);
				Internal.FB.Halt.ShHalt.Execute := TRUE;

				IF Internal.FB.Halt.ShHalt.Error THEN
					Internal.FB.Halt.ShHalt.Execute := FALSE;
					ErrorID := Internal.FB.Halt.ShHalt.ErrorID;
					Internal.State := rdi_ERROR;
				ELSIF Internal.FB.Halt.ShHalt.Done THEN
					Internal.FB.Halt.ShHalt.Execute := FALSE;
					Internal.State := rdi_WAIT_FOR_COMMAND;
				END_IF

			rdi_ASM_LEVITATION:
				CurrentState := 'rdi_ASM_LEVITATION';
				Internal.FB.Levitation.AsmLevitation.Parameters := Parameters.Levitation;
				Internal.FB.Levitation.AsmLevitation.Execute := TRUE;

				IF Internal.FB.Levitation.AsmLevitation.Error THEN
					Internal.FB.Levitation.AsmLevitation.Execute := FALSE;
					ErrorID := Internal.FB.Levitation.AsmLevitation.ErrorID;
					Internal.State := rdi_ERROR;
				ELSIF Internal.FB.Levitation.AsmLevitation.Acknowledge THEN
					Internal.FB.Levitation.AsmLevitation.Execute := FALSE;
					Internal.State := rdi_WAIT_FOR_COMMAND;
				END_IF

			rdi_SHUTTLE_LEVITATION:
				CurrentState := 'rdi_SHUTTLE_LEVITATION';
				Internal.FB.Levitation.ShLevitation.Shuttle := ADR(Internal.Status.SelectedShuttleAxis);
				Internal.FB.Levitation.ShLevitation.Parameters := Parameters.Levitation;
				Internal.FB.Levitation.ShLevitation.Execute := TRUE;

				IF Internal.FB.Levitation.ShLevitation.Error THEN
					Internal.FB.Levitation.ShLevitation.Execute := FALSE;
					ErrorID := Internal.FB.Levitation.ShLevitation.ErrorID;
					Internal.State := rdi_ERROR;
				ELSIF Internal.FB.Levitation.ShLevitation.Acknowledge THEN
					Internal.FB.Levitation.ShLevitation.Execute := FALSE;
					Internal.State := rdi_WAIT_FOR_COMMAND;
				END_IF

			rdi_ASM_BUFFER:
				CurrentState := 'rdi_ASM_BUFFER';
				Internal.FB.Buffer.AsmBuffer.Option := Parameters.Buffer;
				Internal.FB.Buffer.AsmBuffer.Execute := TRUE;

				IF Internal.FB.Buffer.AsmBuffer.Error THEN
					Internal.FB.Buffer.AsmBuffer.Execute := FALSE;
					ErrorID := Internal.FB.Buffer.AsmBuffer.ErrorID;
					Internal.State := rdi_ERROR;
				ELSIF Internal.FB.Buffer.AsmBuffer.Done THEN
					Internal.FB.Buffer.AsmBuffer.Execute := FALSE;
					Internal.State := rd_SHUTTLE_BUFFER_STATUS;
				END_IF

			rdi_SHUTTLE_BUFFER:
				CurrentState := 'rdi_SHUTTLE_BUFFER';
				Internal.FB.Buffer.ShBuffer.Shuttle := ADR(Internal.Status.SelectedShuttleAxis);
				Internal.FB.Buffer.ShBuffer.Option := Parameters.Buffer;
				Internal.FB.Buffer.ShBuffer.Execute := TRUE;

				IF Internal.FB.Buffer.ShBuffer.Error THEN
					Internal.FB.Buffer.ShBuffer.Execute := FALSE;
					ErrorID := Internal.FB.Buffer.ShBuffer.ErrorID;
					Internal.State := rdi_ERROR;
				ELSIF Internal.FB.Buffer.ShBuffer.Done THEN
					Internal.FB.Buffer.ShBuffer.Execute := FALSE;
					Internal.State := rd_SHUTTLE_BUFFER_STATUS;
				END_IF

			rd_SHUTTLE_BUFFER_STATUS:
				CurrentState := 'rd_SHUTTLE_BUFFER_STATUS';
				Internal.FB.Buffer.ShBuffer.Shuttle := ADR(Internal.Status.SelectedShuttleAxis);
				Internal.FB.Buffer.ShBuffer.Option := mcACP6D_BUFFER_GET_STATUS;
				Internal.FB.Buffer.ShBuffer.Execute := TRUE;

				IF Internal.FB.Buffer.ShBuffer.Error THEN
					Internal.FB.Buffer.ShBuffer.Execute := FALSE;
					ErrorID := Internal.FB.Buffer.ShBuffer.ErrorID;
					Internal.State := rdi_ERROR;
				ELSIF Internal.FB.Buffer.ShBuffer.Done THEN
					ShuttleBufferInfo.ShuttleID := ShuttleID;
					ShuttleBufferInfo.NumberOfCommands := Internal.FB.Buffer.ShBuffer.BufferInfo.NumberOfCommands;
					ShuttleBufferInfo.State := Internal.FB.Buffer.ShBuffer.BufferInfo.State;
					Internal.FB.Buffer.ShBuffer.Execute := FALSE;
					Internal.State := rdi_WAIT_FOR_COMMAND;
				END_IF

			rdi_SHUTTLE_RECOVER:
				CurrentState := 'rdi_SHUTTLE_RECOVER';
				Internal.FB.Shuttle.ShRecover.Shuttle := ADR(Internal.Status.SelectedShuttleAxis);

				Internal.FB.Shuttle.ShRecover.Execute := TRUE;

				IF Internal.FB.Shuttle.ShRecover.Error THEN
					Internal.FB.Shuttle.ShRecover.Execute := FALSE;
					ErrorID := Internal.FB.Shuttle.ShRecover.ErrorID;
					Internal.State := rdi_ERROR;
				ELSIF Internal.FB.Shuttle.ShRecover.Done THEN
					Internal.FB.Shuttle.ShRecover.Execute := FALSE;
					Internal.State := rdi_WAIT_FOR_COMMAND;
				END_IF

			rdi_ASM_REBOOT:
				CurrentState := 'rdi_ASM_REBOOT';
				Internal.FB.Asm.AsmReboot.Execute := TRUE;

				IF Internal.FB.Asm.AsmReboot.Error THEN
					Internal.FB.Asm.AsmReboot.Execute := FALSE;
					ErrorID := Internal.FB.Asm.AsmReboot.ErrorID;
					Internal.State := rdi_ERROR;
				ELSIF Internal.FB.Asm.AsmReadStatus.AssemblyDisabled THEN
					Internal.FB.Asm.AsmReboot.Execute := FALSE;
					Internal.State := rdi_WAIT_FOR_POWER_ON;
				END_IF

			rdi_POWER_OFF:
				CurrentState := 'rdi_POWER_OFF';
				Internal.FB.Asm.AsmPowerOff.Execute := TRUE;

				IF Internal.FB.Asm.AsmPowerOff.Error THEN
					Internal.FB.Asm.AsmPowerOff.Execute := FALSE;
					ErrorID := Internal.FB.Asm.AsmPowerOff.ErrorID;
					Internal.State := rdi_ERROR;
				ELSIF Internal.FB.Asm.AsmReadStatus.AssemblyDisabled THEN

					Internal.FB.Asm.AsmPowerOff.Execute := FALSE;
					Internal.State := rdi_WAIT_FOR_POWER_ON;
				END_IF

			rdi_ERROR:
				CurrentState := 'rdi_ERROR';
				Error := TRUE;

				IF EDGEPOS(ErrorReset) THEN
					Error := FALSE;
					ErrorID := 0;
					Internal.State := rdi_WAIT_FOR_COMMAND;
				END_IF

		END_CASE

		(* FB calls *)
		Internal.FB.Asm.AsmReadStatus();
		Internal.FB.Asm.AsmGetInfo();
		Internal.FB.Asm.AsmGetShuttle();
		Internal.FB.Asm.AsmPowerOn();
		Internal.FB.Asm.AsmPowerOff();
		Internal.FB.Asm.AsmReboot();

		Internal.FB.Move.Linear();
		Internal.FB.Move.Arc();
		Internal.FB.Move.Short();
		Internal.FB.Move.SixDOF();
		Internal.FB.Move.Async();

		Internal.FB.Stop.AsmStop();
		Internal.FB.Stop.ShStop();
		Internal.FB.Halt.AsmHalt();
		Internal.FB.Halt.ShHalt();

		Internal.FB.Levitation.AsmLevitation();
		Internal.FB.Levitation.ShLevitation();
		Internal.FB.Buffer.AsmBuffer();
		Internal.FB.Buffer.ShBuffer();

		Internal.FB.Shuttle.ShRecover();

		(* set the output statuses *)
		Active := Enable;
		PowerOn := Internal.FB.Asm.AsmReadStatus.AssemblyReady;

		AsmStatus.AssemblyDisabled := Internal.FB.Asm.AsmReadStatus.AssemblyDisabled;
		AsmStatus.AssemblyErrorStop := Internal.FB.Asm.AsmReadStatus.AssemblyErrorStop;
		AsmStatus.AssemblyHoming := Internal.FB.Asm.AsmReadStatus.AssemblyHoming;
		AsmStatus.AssemblyReady := Internal.FB.Asm.AsmReadStatus.AssemblyReady;
		AsmStatus.AssemblyStartUp := Internal.FB.Asm.AsmReadStatus.AssemblyStartUp;
		AsmStatus.AssemblyStopping := Internal.FB.Asm.AsmReadStatus.AssemblyStopping;

		(* cyclically update shuttle info *)
		MovementActive := FALSE;

		FOR i := 0 TO MAX_NUM_SHUTTLES_M1 DO
			Internal.FB.Shuttle.ShReadInfo[i]();

			IF Internal.FB.Shuttle.ShReadInfo[i].Valid THEN
				ShuttleArray[i].ShuttleID := Internal.FB.Shuttle.ShReadInfo[i].ShuttleInfo.ShuttleID;
				ShuttleArray[i].Position := Internal.FB.Shuttle.ShReadInfo[i].ShuttleInfo.Position;
				ShuttleArray[i].State := Internal.FB.Shuttle.ShReadInfo[i].ShuttleInfo.State;

				MovementActive := MovementActive OR (ShuttleArray[i].State = mcACP6D_SH_STATE_MOTION) OR (ShuttleArray[i].State = mcACP6D_SH_STATE_STOPPING) OR (ShuttleArray[i].State = mcACP6D_SH_STATE_OBSTACLE);
			END_IF

		END_FOR

		(* if not enabled *)
	ELSE

	END_IF

END_FUNCTION_BLOCK
```

### Library Logical/Libraries/Acp6dHlpr (IEC)

#### Types.typ - Exported data types
```iecst
TYPE
	Acp6dMoveBlockParsTyp : 	STRUCT
		NumMoves : USINT;
		MoveList : REFERENCE TO ARRAY[0..1]OF Acp6DMoveListTyp;
	END_STRUCT;
	Acp6DMoveTypeEnum :
		(
		acp6d_MOVE_LINEAR,
		acp6d_MOVE_ARC,
		acp6d_MOVE_SHORT,
		acp6d_MOVE_PAUSE
		);
	Acp6DMoveListTyp : 	STRUCT
		MoveType : Acp6DMoveTypeEnum;
		Linear : McAcp6DInPlaneParType;
		Arc : McAcp6DArcParType;
		ShortAxis : McAcp6DShortAxParType;
		PauseTime : TIME;
	END_STRUCT;
	Acp6DMoveBlockInternalTyp : 	STRUCT
		state : Acp6dMoveStatesEnum;
		errorState : Acp6dMoveStatesEnum;
		currentIndex : UINT;
		numMoves : USINT;
		movesList : ARRAY[0..maxMOVES_ARRAY]OF Acp6DMoveListTyp;
		fbs : Acp6DMoveInternalFbsTYp;
	END_STRUCT;
	Acp6DMoveInternalFbsTYp : 	STRUCT
		LinearFb : MC_BR_MoveInPlane_Acp6D;
		ArcFb : MC_BR_MoveArc_Acp6D;
		ShortAxFb : MC_BR_MoveShortAxis_Acp6D;
		PauseFb : TON;
	END_STRUCT;
	Acp6dMoveStatesEnum :
		(
		MV_INIT,
		MV_CHECK_CMD,
		MV_CHECK_FOR_LAST,
		MV_MOVE_LINEAR,
		MV_MOVE_ARC,
		MV_MOVE_SHORT,
		MV_PAUSE,
		MV_WAIT_FOR_LAST,
		MV_DONE,
		MV_ERROR,
		MV_RESET
		);
END_TYPE
```

#### Constants.var - Exported constants
```iecst
VAR CONSTANT
	maxMOVES : USINT := 15;
	maxMOVES_ARRAY : USINT := maxMOVES - 1;
END_VAR
```

#### Acp6dHlpr.fun - Exported functions and function blocks
```iecst
FUNCTION_BLOCK Acp6DMoveBlockFb
	VAR_INPUT
		Execute : BOOL;
		Shuttle : {REDUND_UNREPLICABLE} Mc6DShuttleType;
		Pars : Acp6dMoveBlockParsTyp;
		WaitForLast : BOOL;
	END_VAR
	VAR_OUTPUT
		Busy : BOOL;
		Error : BOOL;
		ErrorID : UDINT;
		WaitingForLast : BOOL;
		Done : BOOL;
	END_VAR
	VAR
		internal : Acp6DMoveBlockInternalTyp;
	END_VAR
END_FUNCTION_BLOCK
```

#### Acp6DMoveBlockFb.st
```iecst
(* TODO: Add your comment here *)
FUNCTION_BLOCK Acp6DMoveBlockFb

	CASE internal.state OF
		// ***************************** Init State
		MV_INIT:
			IF Execute THEN
				IF Pars.NumMoves > maxMOVES THEN
					internal.errorState := internal.state;
					internal.state := MV_ERROR;
					Error := TRUE;
					ErrorID := -1;
				ELSIF Pars.NumMoves = 0 THEN
					Done := TRUE;
					internal.state := MV_DONE;
				ELSE
					internal.currentIndex := 0;
					internal.numMoves := Pars.NumMoves;
					brsmemcpy(ADR(internal.movesList),Pars.MoveList,internal.numMoves * SIZEOF(internal.movesList[0]));
					internal.state := MV_CHECK_CMD;
				END_IF
			ELSE
				Error := FALSE;
				ErrorID := 0;
				WaitingForLast := FALSE;
				Done := FALSE;
			END_IF

		// ***************************** Checking Cmd of Current Parameter
		MV_CHECK_CMD:
			IF internal.currentIndex = internal.numMoves THEN
				IF WaitForLast THEN
					internal.state := MV_WAIT_FOR_LAST;
				ELSE
				Done := TRUE;
					internal.state := MV_DONE;
				END_IF
			ELSE
				CASE internal.movesList[internal.currentIndex].MoveType OF
					acp6d_MOVE_LINEAR:
						internal.fbs.LinearFb.Shuttle := ADR(Shuttle);
						internal.fbs.LinearFb.Parameters := internal.movesList[internal.currentIndex].Linear;
						internal.fbs.LinearFb.Execute := TRUE;

						internal.state := MV_MOVE_LINEAR;
					acp6d_MOVE_ARC:
						internal.fbs.ArcFb.Shuttle := ADR(Shuttle);
						internal.fbs.ArcFb.Parameters := internal.movesList[internal.currentIndex].Arc;
						internal.fbs.ArcFb.Execute := TRUE;

						internal.state := MV_MOVE_ARC;
					acp6d_MOVE_SHORT:
						internal.fbs.ShortAxFb.Shuttle := ADR(Shuttle);
						internal.fbs.ShortAxFb.Parameters := internal.movesList[internal.currentIndex].ShortAxis;
						internal.fbs.ShortAxFb.Execute := TRUE;

						internal.state := MV_MOVE_SHORT;
					acp6d_MOVE_PAUSE:
						internal.fbs.PauseFb.IN := TRUE;
						internal.fbs.PauseFb.PT := internal.movesList[internal.currentIndex].PauseTime;
						internal.state := MV_PAUSE;
				END_CASE;
				WaitingForLast := (internal.currentIndex + 1) = internal.numMoves AND WaitForLast;
			END_IF
		// ***************************** Linear Move State
		MV_MOVE_LINEAR:
			IF internal.fbs.LinearFb.Error THEN
				internal.errorState := internal.state;
				internal.state := MV_ERROR;
				Error := TRUE;
				ErrorID := internal.fbs.LinearFb.ErrorID;
			ELSIF internal.fbs.LinearFb.Acknowledge THEN
				internal.fbs.LinearFb.Execute := FALSE OR WaitingForLast;
				internal.currentIndex := internal.currentIndex + 1;

				internal.state := MV_CHECK_CMD;
			END_IF

		// ***************************** Arc Move State
		MV_MOVE_ARC:
			IF internal.fbs.ArcFb.Error THEN
				internal.errorState := internal.state;
				internal.state := MV_ERROR;
				Error := TRUE;
				ErrorID := internal.fbs.ArcFb.ErrorID;
			ELSIF internal.fbs.ArcFb.Acknowledge THEN
				internal.fbs.ArcFb.Execute := FALSE OR WaitingForLast;
				internal.currentIndex := internal.currentIndex + 1;

				internal.state := MV_CHECK_CMD;
			END_IF
		// ***************************** Short Axis Move State
		MV_MOVE_SHORT:
			IF internal.fbs.ShortAxFb.Error THEN
				internal.errorState := internal.state;
				internal.state := MV_ERROR;
				Error := TRUE;
				ErrorID := internal.fbs.ShortAxFb.ErrorID;
			ELSIF internal.fbs.ShortAxFb.Acknowledge THEN
				internal.fbs.ShortAxFb.Execute := FALSE OR WaitingForLast;
				internal.currentIndex := internal.currentIndex + 1;

				internal.state := MV_CHECK_CMD;
			END_IF
		// ***************************** Pause Move State
		MV_PAUSE:
			IF internal.fbs.PauseFb.Q THEN
				internal.fbs.PauseFb.IN := FALSE;
				internal.currentIndex := internal.currentIndex + 1;

				internal.state := MV_CHECK_CMD;
			END_IF
		// ***************************** Waiting for the last command State
		MV_WAIT_FOR_LAST:
			CASE internal.movesList[internal.currentIndex - 1].MoveType OF
				acp6d_MOVE_LINEAR:
					IF internal.fbs.LinearFb.Done THEN
						internal.fbs.LinearFb.Execute := FALSE;
						WaitingForLast := FALSE;
						Done := TRUE;
						internal.state := MV_DONE;
					END_IF
				acp6d_MOVE_ARC:
					IF internal.fbs.ArcFb.Done THEN
						internal.fbs.ArcFb.Execute := FALSE;
						WaitingForLast := FALSE;
						Done := TRUE;
						internal.state := MV_DONE;
					END_IF
				acp6d_MOVE_SHORT:
					IF internal.fbs.ShortAxFb.Done THEN
						internal.fbs.ShortAxFb.Execute := FALSE;
						WaitingForLast := FALSE;
						Done := TRUE;
						internal.state := MV_DONE;
					END_IF
				acp6d_MOVE_PAUSE:
					WaitingForLast := FALSE;
					Done := TRUE;
					internal.state := MV_DONE;

			END_CASE;
		// ***************************** Done State
		MV_DONE:
			IF NOT Execute THEN
				internal.state := MV_RESET;
			END_IF
		// ***************************** Error State
		MV_ERROR:
			IF NOT Execute THEN
				internal.state := MV_RESET;
			END_IF
		// ***************************** Reset State
		MV_RESET:
			WaitingForLast := FALSE;
			Error := FALSE;
			ErrorID := 0;
			Done := FALSE;

			internal.currentIndex := 0;
			internal.numMoves := 0;
			brsmemset(ADR(internal.movesList),0,internal.numMoves * SIZEOF(internal.movesList[0]));

			internal.fbs.LinearFb.Execute := FALSE;
			internal.fbs.ArcFb.Execute := FALSE;
			internal.fbs.ShortAxFb.Execute := FALSE;
			internal.fbs.PauseFb.IN := FALSE;

			internal.state := MV_INIT;

	END_CASE

	//FB Calls
	internal.fbs.LinearFb();
	internal.fbs.ArcFb();
	internal.fbs.ShortAxFb();
	internal.fbs.PauseFb();

END_FUNCTION_BLOCK
```

### Library Logical/Libraries/Router6D (ANSIC)
Depends on: McAcp6D, AsSem, ArEventLog

#### Types.typ - Router Types
```iecst
TYPE
	rl6dPositionType : 	STRUCT  (*Position on ACOPOS 6D Assembly*)
		X : REAL := 0; (*X Position*)
		Y : REAL := 0; (*Y Position*)
	END_STRUCT;
	rl6dRouterType : 	STRUCT  (*Router handle*)
		Ident : UDINT := 0; (*Router Ident*)
	END_STRUCT;
	rl6dPathType : 	STRUCT  (*Path handle*)
		Ident : UDINT := 0; (*Path Ident*)
	END_STRUCT;
	rl6dDestinationType : 	STRUCT  (*Destination handle*)
		Ident : UDINT := 0; (*Destination Ident*)
	END_STRUCT;
	rl6dWaypointType : 	STRUCT  (*Waypoint handle*)
		Ident : UDINT; (*Waypoint Ident*)
	END_STRUCT;
	rl6dShuttleType : 	STRUCT  (*Shuttle handle*)
		Ident : UDINT := 0; (*Shuttle Ident*)
	END_STRUCT;
	rl6dRouterManInternalType : 	STRUCT  (*Internal Data*)
		State : USINT := 0; (*Router state*)
	END_STRUCT;
	rl6dRouterAddPathInternalType : 	STRUCT  (*Internal Data*)
		State : USINT := 0; (*FB state*)
		Reference : UDINT := 0; (*Reference*)
	END_STRUCT;
	rl6dGetPathInternalType : 	STRUCT  (*Internal Data*)
		State : USINT := 0; (*FB state*)
		DataAddress : UDINT := 0; (*Recorded Data Address*)
		DataSize : UDINT := 0; (*Recorded Data Size*)
	END_STRUCT;
	rl6dRouterAddDestInternalType : 	STRUCT  (*Internal Data*)
		State : USINT := 0; (*FB state*)
		Reference : UDINT := 0; (*Reference*)
	END_STRUCT;
	rl6dDestAddRecPosInternalType : 	STRUCT  (*Internal Data*)
		State : USINT := 0; (*FB state*)
	END_STRUCT;
	rl6dDestSetWaypntInternalType : 	STRUCT  (*Internal Data*)
		State : USINT := 0; (*FB state*)
	END_STRUCT;
	rl6dRouterAddWaypntInternalType : 	STRUCT  (*Internal Data*)
		State : USINT := 0; (*FB state*)
		Reference : UDINT := 0; (*Reference*)
	END_STRUCT;
	rl6dWaypointAddDestInternalType : 	STRUCT  (*Internal Data*)
		State : USINT := 0; (*FB state*)
	END_STRUCT;
	rl6dWaypntSetWaypntInternalType : 	STRUCT  (*Internal Data*)
		State : USINT := 0; (*FB state*)
	END_STRUCT;
	rl6dRtrAddShFromAsmInternalType : 	STRUCT  (*Internal Data*)
		State : USINT := 0; (*State of execution*)
	END_STRUCT;
	rl6dRecoverModeEnum :
		( (*Method to use for recovery*)
		rl6dRECOVER_MODE_BASIC (*Basic recover mode*)
		);
	rl6dDestinationMonInternalType : 	STRUCT  (*Internal Data*)
		State : USINT := 0; (*FB state*)
		Reference : UDINT := 0; (*Reference*)
	END_STRUCT;
	rl6dShMoveDestInternalType : 	STRUCT  (*Internal Data*)
		State : USINT := 0; (*FB state*)
		Reference : UDINT := 0; (*Reference*)
	END_STRUCT;
	rl6dShCopyUserDataInternalType : 	STRUCT  (*Internal Data*)
		State : USINT;
	END_STRUCT;
	rl6dShCopyUserDataModeEnum :
		( (*Mode of shuttle copy user data*)
		rl6dSH_COPY_USER_DATA_READ, (*Read user data*)
		rl6dSH_COPY_USER_DATA_WRITE (*Write user data*)
		);
END_TYPE
```

#### Variables.var - Router Constants
```iecst
(*Constants*)
VAR CONSTANT
	rl6dMAX_RECOVER_SHUTTLES : USINT := 79; (*Maximum number of shuttles that can be recovered in one pass*)
END_VAR
(*Type IDs*)
VAR CONSTANT
	rl6dNO_TYPE_ID : UDINT := 0; (*The object is invalid*)
	rl6dROUTER_TYPE_ID : UDINT := 1003478341; (*The object is a router*)
	rl6dSEM_MAN_TYPE_ID : UDINT := 435837; (*The object is a sem man*)
	rl6dROUTER_SEM_TYPE_ID : UDINT := 235; (*The object is a router sem*)
	rl6dDESTINATION_TYPE_ID : UDINT := 439482759; (*The object is a destination*)
	rl6dDESTINATION_IF_TYPE_ID : UDINT := 19827452; (*The object is a destination interface*)
	rl6dPATH_TYPE_ID : UDINT := 971846639; (*The object is a path*)
	rl6dWAYPOINT_TYPE_ID : UDINT := 72341095; (*The object is a waypoint*)
	rl6dSHUTTLE_TYPE_ID : UDINT := 32490572; (*The object is a shuttle*)
	rl6dSHUTTLE_IF_TYPE_ID : UDINT := 579822341; (*The object is a shuttle interface*)
END_VAR
(*Heap*)
VAR CONSTANT
	rl6dHEAP_SIZE : UDINT := 16#FFFFF; (*Heap size*)
END_VAR
(*Errors*)
VAR CONSTANT
	rl6dERR_NULL_POINTER : DINT := -535887871; (*The pointer is a null pointer*)
	rl6dERR_ROUTER_INVALID : DINT := -535887870; (*The router reference is invalid*)
	rl6dERR_SEM_MAN_INVALID : DINT := -535887869; (*The semaphore manager reference is invalid*)
	rl6dERR_ROUTER_SEM_INVALID : DINT := -535887868; (*The router semaphore reference is invalid*)
	rl6dERR_DESTINATION_INVALID : DINT := -535887867; (*The destination reference is invalid*)
	rl6dERR_DESTINATION_IF_INVALID : DINT := -535887866; (*The destination interface reference is invalid*)
	rl6dERR_PATH_INVALID : DINT := -535887865; (*The path reference is invalid*)
	rl6dERR_SHUTTLE_INVALID : DINT := -535887864; (*The shuttle reference is invalid*)
	rl6dERR_SHUTTLE_IF_INVALID : DINT := -535887863; (*The shuttle interface reference is invalid*)
	rl6dERR_WAYPOINT_INVALID : DINT := -535887862; (*The waypoint interface reference is invalid*)
	rl6dERR_USER_DATA_SIZE_ZERO : DINT := -535887772; (*The user data must be greater than zero bytes*)
	rl6dERR_USER_DATA_SIZE_MISMATCH : DINT := -535887771; (*The size of the user data does not match that defined for the router*)
	rl6dERR_USER_DATA_NULL_POINTER : DINT := -53588777; (*The address of the User Data is set to null*)
	rl6dERR_DATA_ALIGNMENT : DINT := -535887672; (*The size of the input data does not match the size of an array of the expected datatype*)
	rl6dERR_OBJ_NAME_EXISTS : DINT := -535887572; (*The name of this type of object already exists*)
	rl6dERR_NO_OBJ_NAME : DINT := -535887571; (*No name was given for the new object*)
	rl6dERR_SHUTTLE : DINT := -535887472; (*Shuttle encountered an error*)
	rl6dERR_GET_SHUTTLES : DINT := -535887471; (*Get shuttles on assembly encountered an error*)
	rl6dERR_MOVE_IN_PLANE_ASYNC : DINT := -535887470; (*Move in plane async encountered an error*)
END_VAR
(*Info*)
VAR CONSTANT
	rl6dINFO_ROUTED_MOVE_START : DINT := 1611595786; (*A routed move has started*)
	rl6dINFO_DIRECT_MOVE_START : DINT := 1611595787; (*A direct move has started*)
	rl6dINFO_MOVE_PATH_START : DINT := 1611595788; (*Move along a path has started*)
	rl6dINFO_MOVE_WAYPOINT : DINT := 1611595789; (*A move to a waypoint has started*)
	rl6dINFO_ROUTED_MOVE_WAYPOINT : DINT := 1611595790; (*A routed move has started via a specified waypoint*)
	rl6dINFO_DESTINATION_ARRIVE : DINT := 1611595796; (*A shuttle has arrived at a destination*)
	rl6dINFO_DESTINATION_UPDATE : DINT := 1611595797; (*A shuttle route destination has been changed*)
	rl6dINFO_GET_SHUTTLES_START : DINT := 1611595806; (*Router has started to get shuttles on the assembly*)
	rl6dINFO_GET_SHUTTLES_DONE : DINT := 1611595807; (*Router has completed getting shuttles on the assembly*)
	rl6dINFO_RECOVERY_START : DINT := 1611595808; (*Router has started recovering shuttles*)
	rl6dINFO_RECOVERY_DONE : DINT := 1611595809; (*Router has completed recovering shuttles*)
	rl6dINFO_RECOVERY_ASSIGNMENT : DINT := 1611595810; (*Router has assigned a shuttle during recovery*)
END_VAR
```
